C07281=1079.197,-43.335,442.916,173.632,20.227,153.492
C07282=1079.203,-43.085,442.903,173.633,20.229,153.493
C07283=1079.210,-42.836,442.891,173.635,20.230,153.493
C07284=1079.215,-42.586,442.879,173.636,20.232,153.493
C07285=1079.221,-42.337,442.866,173.637,20.234,153.493
C07286=1079.228,-42.087,442.854,173.639,20.236,153.493
C07287=1079.233,-41.837,442.842,173.640,20.238,153.493
C07288=1079.239,-41.588,442.830,173.642,20.240,153.493
C07289=1079.245,-41.338,442.817,173.644,20.242,153.493
C07290=1079.251,-41.088,442.805,173.645,20.244,153.494
C07291=1079.257,-40.839,442.793,173.646,20.246,153.494
C07292=1079.263,-40.589,442.780,173.648,20.248,153.494
C07293=1079.269,-40.340,442.769,173.649,20.250,153.494
C07294=1079.275,-40.090,442.756,173.650,20.252,153.494
C07295=1079.281,-39.840,442.743,173.652,20.253,153.494
C07296=1079.288,-39.590,442.731,173.653,20.255,153.494
C07297=1079.293,-39.341,442.719,173.655,20.258,153.494
C07298=1079.299,-39.091,442.707,173.657,20.260,153.495
C07299=1079.305,-38.842,442.694,173.658,20.262,153.495
C07300=1079.311,-38.592,442.682,173.659,20.263,153.495
C07301=1079.317,-38.342,442.670,173.661,20.265,153.495
C07302=1079.323,-38.093,442.657,173.662,20.267,153.495
C07303=1079.329,-37.843,442.645,173.663,20.269,153.495
C07304=1079.334,-37.593,442.632,173.665,20.272,153.495
C07305=1079.340,-37.343,442.620,173.667,20.274,153.496
C07306=1079.346,-37.094,442.608,173.668,20.276,153.496
C07307=1079.353,-36.845,442.595,173.669,20.278,153.496
C07308=1079.359,-36.595,442.582,173.671,20.279,153.496
C07309=1079.364,-36.345,442.570,173.672,20.281,153.496
C07310=1079.370,-36.096,442.558,173.673,20.283,153.496
C07311=1079.376,-35.846,442.545,173.674,20.285,153.496
C07312=1079.382,-35.596,442.533,173.677,20.288,153.497
C07313=1079.388,-35.347,442.520,173.678,20.290,153.497
C07314=1079.393,-35.097,442.507,173.679,20.292,153.497
C07315=1079.399,-34.848,442.495,173.680,20.294,153.497
C07316=1079.406,-34.599,442.483,173.682,20.296,153.497
C07317=1079.412,-34.349,442.470,173.683,20.298,153.497
C07318=1079.417,-34.099,442.457,173.685,20.300,153.497
C07319=1079.423,-33.849,442.445,173.687,20.302,153.498
C07320=1079.430,-33.575,442.431,173.688,20.304,153.498
C07321=1079.436,-33.302,442.417,173.689,20.306,153.498
C07322=1079.442,-33.028,442.404,173.691,20.309,153.498
C07323=1079.449,-32.754,442.390,173.692,20.311,153.498
C07324=1079.455,-32.504,442.376,173.694,20.313,153.499
C07325=1079.461,-32.254,442.364,173.695,20.315,153.499
C07326=1079.467,-32.004,442.351,173.697,20.317,153.499
C07327=1079.473,-31.755,442.339,173.699,20.318,153.499
C07328=1079.479,-31.505,442.325,173.700,20.320,153.499
C07329=1079.484,-31.256,442.313,173.701,20.322,153.499
C07330=1079.491,-31.007,442.301,173.703,20.324,153.499
C07331=1079.497,-30.757,442.288,173.704,20.326,153.500
C07332=1079.503,-30.507,442.275,173.705,20.328,153.500
C07333=1079.509,-30.258,442.263,173.707,20.331,153.500
C07334=1079.515,-30.008,442.250,173.709,20.333,153.500
C07335=1079.521,-29.758,442.237,173.710,20.335,153.500
C07336=1079.527,-29.509,442.225,173.711,20.337,153.500
C07337=1079.532,-29.259,442.212,173.712,20.339,153.500
C07338=1079.538,-29.010,442.199,173.714,20.341,153.501
C07339=1079.544,-28.760,442.187,173.716,20.343,153.501
C07340=1079.550,-28.510,442.174,173.717,20.345,153.501
C07341=1079.556,-28.261,442.161,173.719,20.347,153.501
C07342=1079.562,-28.011,442.148,173.720,20.349,153.501
C07343=1079.568,-27.761,442.136,173.721,20.351,153.501
C07344=1079.574,-27.512,442.122,173.722,20.353,153.501
C07345=1079.580,-27.262,442.110,173.725,20.355,153.502
C07346=1079.587,-27.013,442.097,173.726,20.357,153.502
C07347=1079.592,-26.763,442.084,173.727,20.359,153.502
C07348=1079.598,-26.513,442.071,173.728,20.361,153.502
C07349=1079.604,-26.264,442.058,173.730,20.363,153.502
C07350=1079.609,-26.014,442.045,173.731,20.365,153.502
C07351=1079.615,-25.765,442.032,173.733,20.368,153.503
C07352=1079.621,-25.515,442.020,173.734,20.370,153.503
C07353=1079.627,-25.266,442.006,173.736,20.372,153.503
C07354=1079.633,-25.016,441.994,173.737,20.374,153.503
C07355=1079.639,-24.766,441.981,173.738,20.376,153.503
C07356=1079.645,-24.517,441.967,173.739,20.378,153.504
C07357=1079.651,-24.267,441.955,173.742,20.381,153.504
C07358=1079.657,-24.017,441.941,173.743,20.383,153.504
C07359=1079.663,-23.768,441.929,173.744,20.385,153.504
C07360=1079.668,-23.518,441.915,173.745,20.387,153.504
C07361=1079.674,-23.268,441.903,173.747,20.389,153.504
C07362=1079.680,-23.020,441.890,173.748,20.391,153.504
C07363=1079.686,-22.770,441.877,173.750,20.393,153.505
C07364=1079.692,-22.520,441.864,173.751,20.395,153.505
C07365=1079.697,-22.270,441.851,173.753,20.397,153.505
C07366=1079.703,-22.021,441.837,173.754,20.399,153.505
C07367=1079.709,-21.771,441.825,173.755,20.401,153.505
C07368=1079.715,-21.522,441.812,173.757,20.403,153.505
C07369=1079.722,-21.273,441.798,173.759,20.405,153.506
C07370=1079.727,-21.022,441.785,173.760,20.407,153.506
C07371=1079.733,-20.773,441.772,173.761,20.409,153.506
C07372=1079.739,-20.523,441.759,173.763,20.411,153.506
C07373=1079.745,-20.274,441.746,173.764,20.413,153.506
C07374=1079.751,-20.024,441.732,173.766,20.416,153.507
C07375=1079.757,-19.774,441.720,173.767,20.418,153.507
C07376=1079.763,-19.525,441.706,173.768,20.420,153.507
C07377=1079.769,-19.275,441.694,173.770,20.422,153.507
C07378=1079.774,-19.026,441.680,173.771,20.424,153.507
C07379=1079.780,-18.776,441.667,173.772,20.426,153.507
C07380=1079.786,-18.527,441.654,173.774,20.429,153.507
C07381=1079.792,-18.277,441.641,173.776,20.431,153.508
C07382=1079.798,-18.028,441.627,173.777,20.433,153.508
C07383=1079.804,-17.778,441.614,173.778,20.435,153.508
C07384=1079.811,-17.503,441.600,173.780,20.437,153.508
C07385=1079.817,-17.228,441.585,173.782,20.440,153.508
C07386=1079.824,-16.953,441.570,173.783,20.442,153.509
C07387=1079.830,-16.679,441.557,173.785,20.444,153.509
C07388=1079.837,-16.429,441.543,173.786,20.446,153.509
C07389=1079.842,-16.180,441.529,173.788,20.448,153.509
C07390=1079.849,-15.930,441.516,173.789,20.450,153.509
C07391=1079.854,-15.680,441.503,173.791,20.453,153.509
C07392=1079.860,-15.431,441.489,173.792,20.455,153.510
C07393=1079.866,-15.182,441.476,173.793,20.457,153.510
C07394=1079.872,-14.932,441.463,173.795,20.459,153.510
C07395=1079.878,-14.682,441.450,173.796,20.461,153.510
C07396=1079.884,-14.433,441.436,173.797,20.463,153.510
C07397=1079.889,-14.183,441.423,173.799,20.465,153.510
C07398=1079.895,-13.934,441.409,173.800,20.468,153.511
C07399=1079.901,-13.684,441.396,173.802,20.470,153.511
C07400=1079.907,-13.435,441.383,173.803,20.472,153.511
C07401=1079.913,-13.185,441.370,173.804,20.474,153.511
C07402=1079.919,-12.936,441.356,173.806,20.476,153.511
C07403=1079.925,-12.686,441.342,173.808,20.478,153.512
C07404=1079.930,-12.436,441.329,173.809,20.481,153.512
C07405=1079.936,-12.187,441.316,173.810,20.483,153.512
C07406=1079.942,-11.937,441.302,173.811,20.485,153.512
C07407=1079.948,-11.687,441.289,173.814,20.487,153.512
C07408=1079.954,-11.438,441.275,173.815,20.489,153.512
C07409=1079.960,-11.189,441.261,173.816,20.491,153.513
C07410=1079.965,-10.938,441.248,173.817,20.494,153.513
C07411=1079.972,-10.689,441.235,173.819,20.496,153.513
C07412=1079.977,-10.440,441.221,173.821,20.498,153.513
C07413=1079.983,-10.190,441.208,173.822,20.500,153.513
C07414=1079.989,-9.941,441.194,173.823,20.502,153.514
C07415=1079.995,-9.691,441.181,173.825,20.504,153.514
C07416=1080.001,-9.441,441.166,173.826,20.507,153.514
C07417=1080.007,-9.192,441.153,173.828,20.509,153.514
C07418=1080.013,-8.942,441.139,173.829,20.511,153.514
C07419=1080.019,-8.693,441.126,173.830,20.513,153.515
C07420=1080.024,-8.443,441.113,173.832,20.515,153.515
C07421=1080.030,-8.193,441.099,173.833,20.517,153.515
C07422=1080.036,-7.944,441.086,173.835,20.520,153.515
C07423=1080.042,-7.694,441.072,173.836,20.522,153.515
C07424=1080.048,-7.445,441.058,173.837,20.524,153.515
C07425=1080.053,-7.195,441.044,173.839,20.526,153.516
C07426=1080.060,-6.946,441.031,173.840,20.528,153.516
C07427=1080.065,-6.696,441.017,173.842,20.530,153.516
C07428=1080.071,-6.447,441.004,173.843,20.533,153.516
C07429=1080.077,-6.197,440.990,173.845,20.535,153.516
C07430=1080.084,-5.947,440.976,173.846,20.537,153.517
C07431=1080.089,-5.698,440.963,173.848,20.539,153.517
C07432=1080.095,-5.448,440.949,173.849,20.541,153.517
C07433=1080.101,-5.199,440.936,173.850,20.544,153.517
C07434=1080.107,-4.949,440.921,173.852,20.546,153.517
C07435=1080.113,-4.699,440.908,173.853,20.548,153.517
C07436=1080.119,-4.450,440.894,173.855,20.550,153.518
C07437=1080.125,-4.201,440.880,173.856,20.552,153.518
C07438=1080.131,-3.952,440.866,173.858,20.554,153.518
C07439=1080.137,-3.701,440.852,173.859,20.557,153.518
C07440=1080.143,-3.452,440.839,173.860,20.559,153.518
C07441=1080.148,-3.202,440.825,173.862,20.561,153.519
C07442=1080.154,-2.953,440.811,173.864,20.563,153.519
C07443=1080.160,-2.704,440.798,173.865,20.566,153.519
C07444=1080.166,-2.453,440.784,173.866,20.568,153.519
C07445=1080.172,-2.204,440.770,173.868,20.570,153.519
C07446=1080.177,-1.954,440.756,173.869,20.572,153.519
C07447=1080.183,-1.705,440.741,173.871,20.575,153.520
C07448=1080.190,-1.429,440.727,173.872,20.577,153.520
C07449=1080.196,-1.153,440.711,173.874,20.580,153.520
C07450=1080.202,-0.875,440.695,173.875,20.582,153.520
C07451=1080.209,-0.600,440.680,173.877,20.585,153.521
C07452=1080.215,-0.350,440.666,173.878,20.587,153.521
C07453=1080.220,-0.100,440.652,173.880,20.589,153.521
C07454=1080.226,0.148,440.638,173.881,20.591,153.521
C07455=1080.232,0.399,440.624,173.883,20.593,153.521
C07456=1080.237,0.648,440.610,173.884,20.595,153.522
C07457=1080.244,0.898,440.597,173.885,20.598,153.522
C07458=1080.249,1.147,440.583,173.887,20.600,153.522
C07459=1080.255,1.396,440.568,173.889,20.602,153.522
C07460=1080.261,1.646,440.554,173.890,20.604,153.522
C07461=1080.266,1.896,440.540,173.891,20.607,153.523
C07462=1080.272,2.146,440.526,173.892,20.609,153.523
C07463=1080.278,2.395,440.512,173.894,20.611,153.523
C07464=1080.284,2.644,440.498,173.896,20.614,153.523
C07465=1080.290,2.894,440.484,173.897,20.616,153.523
C07466=1080.296,3.143,440.469,173.898,20.618,153.524
C07467=1080.301,3.393,440.456,173.900,20.620,153.524
C07468=1080.307,3.643,440.441,173.901,20.623,153.524
C07469=1080.313,3.892,440.428,173.903,20.625,153.524
C07470=1080.319,4.141,440.413,173.904,20.627,153.524
C07471=1080.324,4.391,440.399,173.905,20.629,153.525
C07472=1080.331,4.641,440.385,173.907,20.632,153.525
C07473=1080.337,4.890,440.371,173.909,20.634,153.525
C07474=1080.342,5.139,440.357,173.910,20.636,153.525
C07475=1080.348,5.390,440.343,173.911,20.638,153.525
C07476=1080.354,5.639,440.328,173.913,20.641,153.526
C07477=1080.359,5.888,440.314,173.914,20.643,153.526
C07478=1080.366,6.138,440.299,173.916,20.644,153.526
C07479=1080.371,6.388,440.286,173.917,20.647,153.526
C07480=1080.377,6.637,440.272,173.918,20.649,153.526
C07481=1080.383,6.887,440.257,173.920,20.651,153.527
C07482=1080.389,7.136,440.243,173.921,20.654,153.527
C07483=1080.395,7.385,440.229,173.923,20.656,153.527
C07484=1080.401,7.635,440.215,173.924,20.658,153.527
C07485=1080.407,7.885,440.201,173.926,20.660,153.527
C07486=1080.413,8.134,440.186,173.927,20.663,153.528
C07487=1080.419,8.384,440.172,173.929,20.665,153.528
C07488=1080.424,8.633,440.157,173.930,20.667,153.528
C07489=1080.430,8.883,440.144,173.932,20.669,153.528
C07490=1080.436,9.132,440.129,173.933,20.672,153.528
C07491=1080.442,9.382,440.115,173.934,20.674,153.529
C07492=1080.447,9.631,440.100,173.936,20.676,153.529
C07493=1080.454,9.881,440.086,173.938,20.678,153.529
C07494=1080.459,10.130,440.071,173.939,20.681,153.529
C07495=1080.465,10.380,440.057,173.940,20.683,153.529
C07496=1080.471,10.629,440.042,173.942,20.685,153.530
C07497=1080.477,10.879,440.029,173.944,20.687,153.530
C07498=1080.483,11.128,440.014,173.945,20.690,153.530
C07499=1080.489,11.378,440.000,173.946,20.691,153.530
C07500=1080.496,11.627,439.985,173.947,20.693,153.530
C07501=1080.501,11.877,439.972,173.949,20.695,153.530
C07502=1080.508,12.127,439.957,173.951,20.698,153.531
C07503=1080.513,12.376,439.943,173.952,20.700,153.531
C07504=1080.519,12.625,439.928,173.953,20.702,153.531
C07505=1080.525,12.875,439.913,173.955,20.704,153.531
C07506=1080.531,13.124,439.899,173.957,20.707,153.532
C07507=1080.537,13.374,439.884,173.958,20.709,153.532
C07508=1080.542,13.624,439.871,173.959,20.711,153.532
C07509=1080.549,13.873,439.856,173.960,20.713,153.532
C07510=1080.555,14.122,439.841,173.962,20.716,153.532
C07511=1080.561,14.372,439.827,173.964,20.718,153.532
C07512=1080.566,14.650,439.811,173.965,20.720,153.533
C07513=1080.573,14.929,439.794,173.967,20.723,153.533
C07514=1080.579,15.207,439.778,173.969,20.726,153.533
C07515=1080.586,15.485,439.762,173.970,20.728,153.533
C07516=1080.592,15.735,439.747,173.971,20.731,153.534
C07517=1080.598,15.984,439.732,173.974,20.733,153.534
C07518=1080.604,16.234,439.718,173.975,20.735,153.534
C07519=1080.610,16.483,439.703,173.976,20.737,153.534
C07520=1080.615,16.732,439.689,173.977,20.739,153.534
C07521=1080.621,16.983,439.674,173.979,20.742,153.535
C07522=1080.626,17.232,439.659,173.980,20.744,153.535
C07523=1080.633,17.482,439.644,173.982,20.746,153.535
C07524=1080.639,17.730,439.630,173.983,20.748,153.535
C07525=1080.645,17.981,439.615,173.985,20.751,153.535
C07526=1080.650,18.230,439.600,173.986,20.753,153.536
C07527=1080.656,18.480,439.585,173.988,20.755,153.536
C07528=1080.662,18.729,439.571,173.989,20.757,153.536
C07529=1080.668,18.979,439.556,173.991,20.760,153.536
C07530=1080.674,19.228,439.542,173.992,20.762,153.536
C07531=1080.679,19.478,439.526,173.994,20.764,153.537
C07532=1080.685,19.727,439.512,173.995,20.767,153.537
C07533=1080.692,19.976,439.497,173.997,20.769,153.537
C07534=1080.697,20.226,439.483,173.998,20.771,153.537
C07535=1080.703,20.476,439.467,173.999,20.773,153.537
C07536=1080.708,20.725,439.453,174.001,20.776,153.538
C07537=1080.714,20.974,439.438,174.003,20.778,153.538
C07538=1080.720,21.224,439.423,174.004,20.780,153.538
C07539=1080.725,21.473,439.409,174.005,20.782,153.538
C07540=1080.732,21.723,439.394,174.007,20.785,153.538
C07541=1080.737,21.972,439.379,174.008,20.787,153.539
C07542=1080.743,22.222,439.364,174.010,20.789,153.539
C07543=1080.749,22.471,439.349,174.011,20.791,153.539
C07544=1080.755,22.721,439.334,174.013,20.794,153.539
C07545=1080.760,22.970,439.319,174.014,20.796,153.539
C07546=1080.767,23.220,439.304,174.016,20.798,153.540
C07547=1080.772,23.470,439.289,174.017,20.801,153.540
C07548=1080.778,23.719,439.275,174.019,20.803,153.540
C07549=1080.784,23.969,439.260,174.020,20.805,153.540
C07550=1080.789,24.218,439.245,174.021,20.808,153.541
C07551=1080.796,24.468,439.230,174.023,20.810,153.541
C07552=1080.801,24.717,439.215,174.025,20.812,153.541
C07553=1080.807,24.967,439.200,174.026,20.814,153.541
C07554=1080.813,25.216,439.185,174.027,20.816,153.541
C07555=1080.819,25.466,439.169,174.029,20.819,153.541
C07556=1080.824,25.714,439.155,174.031,20.821,153.542
C07557=1080.831,25.964,439.140,174.032,20.823,153.542
C07558=1080.836,26.214,439.124,174.034,20.826,153.542
C07559=1080.842,26.463,439.110,174.035,20.828,153.542
C07560=1080.849,26.713,439.095,174.036,20.830,153.543
C07561=1080.854,26.962,439.080,174.038,20.832,153.543
C07562=1080.860,27.212,439.065,174.040,20.835,153.543
C07563=1080.866,27.462,439.049,174.041,20.837,153.543
C07564=1080.871,27.711,439.035,174.042,20.839,153.543
C07565=1080.877,27.961,439.019,174.043,20.841,153.544
C07566=1080.883,28.209,439.004,174.045,20.844,153.544
C07567=1080.889,28.459,438.990,174.047,20.846,153.544
C07568=1080.895,28.708,438.974,174.048,20.848,153.544
C07569=1080.901,28.957,438.959,174.050,20.850,153.544
C07570=1080.907,29.207,438.943,174.051,20.853,153.545
C07571=1080.912,29.457,438.928,174.053,20.855,153.545
C07572=1080.918,29.706,438.913,174.054,20.857,153.545
C07573=1080.923,29.956,438.898,174.056,20.860,153.545
C07574=1080.929,30.205,438.883,174.057,20.862,153.545
C07575=1080.935,30.455,438.867,174.058,20.864,153.546
C07576=1080.941,30.735,438.850,174.061,20.867,153.546
C07577=1080.948,31.014,438.833,174.063,20.870,153.546
C07578=1080.954,31.294,438.816,174.064,20.872,153.546
C07579=1080.961,31.574,438.799,174.066,20.874,153.546
C07580=1080.967,31.823,438.784,174.067,20.876,153.547
C07581=1080.972,32.073,438.769,174.068,20.879,153.547
C07582=1080.978,32.321,438.753,174.070,20.881,153.547
C07583=1080.984,32.571,438.738,174.072,20.883,153.547
C07584=1080.990,32.821,438.722,174.073,20.886,153.548
C07585=1080.995,33.070,438.708,174.074,20.888,153.548
C07586=1081.001,33.320,438.692,174.076,20.890,153.548
C07587=1081.008,33.569,438.676,174.077,20.893,153.548
C07588=1081.013,33.818,438.661,174.079,20.895,153.548
C07589=1081.019,34.068,438.646,174.081,20.897,153.548
C07590=1081.025,34.318,438.631,174.082,20.900,153.549
C07591=1081.030,34.567,438.615,174.083,20.902,153.549
C07592=1081.037,34.816,438.600,174.085,20.904,153.549
C07593=1081.042,35.066,438.584,174.087,20.906,153.549
C07594=1081.048,35.315,438.568,174.088,20.908,153.550
C07595=1081.054,35.565,438.554,174.089,20.910,153.550
C07596=1081.060,35.815,438.538,174.091,20.913,153.550
C07597=1081.065,36.064,438.523,174.093,20.915,153.550
C07598=1081.071,36.313,438.507,174.094,20.917,153.550
C07599=1081.077,36.563,438.492,174.096,20.920,153.550
C07600=1081.083,36.813,438.476,174.097,20.922,153.551
C07601=1081.089,37.061,438.461,174.098,20.924,153.551
C07602=1081.094,37.311,438.445,174.101,20.927,153.551
C07603=1081.100,37.561,438.430,174.102,20.929,153.551
C07604=1081.106,37.810,438.414,174.103,20.931,153.552
C07605=1081.112,38.059,438.399,174.104,20.933,153.552
C07606=1081.118,38.309,438.383,174.106,20.936,153.552
C07607=1081.123,38.559,438.367,174.108,20.938,153.552
C07608=1081.129,38.808,438.352,174.109,20.940,153.552
C07609=1081.135,39.057,438.336,174.111,20.943,153.553
C07610=1081.141,39.307,438.321,174.112,20.945,153.553
C07611=1081.146,39.556,438.305,174.114,20.947,153.553
C07612=1081.152,39.806,438.289,174.116,20.950,153.553
C07613=1081.158,40.055,438.274,174.117,20.952,153.553
C07614=1081.163,40.304,438.258,174.118,20.954,153.554
C07615=1081.169,40.554,438.243,174.120,20.957,153.554
C07616=1081.175,40.803,438.227,174.121,20.959,153.554
C07617=1081.181,41.053,438.211,174.123,20.960,153.554
C07618=1081.186,41.302,438.195,174.125,20.963,153.554
C07619=1081.192,41.552,438.180,174.126,20.965,153.555
C07620=1081.198,41.801,438.164,174.127,20.967,153.555
C07621=1081.204,42.051,438.148,174.129,20.970,153.555
C07622=1081.209,42.300,438.133,174.131,20.972,153.555
C07623=1081.215,42.550,438.117,174.132,20.974,153.555
C07624=1081.221,42.799,438.101,174.134,20.977,153.556
C07625=1081.227,43.049,438.086,174.135,20.979,153.556
C07626=1081.233,43.298,438.070,174.137,20.981,153.556
C07627=1081.238,43.547,438.054,174.138,20.983,153.556
C07628=1081.244,43.796,438.038,174.140,20.986,153.556
C07629=1081.250,44.046,438.023,174.141,20.988,153.557
C07630=1081.256,44.296,438.006,174.143,20.990,153.557
C07631=1081.261,44.544,437.990,174.145,20.993,153.557
C07632=1081.267,44.794,437.975,174.146,20.995,153.557
C07633=1081.273,45.044,437.959,174.147,20.997,153.558
C07634=1081.278,45.293,437.943,174.149,21.000,153.558
C07635=1081.284,45.542,437.927,174.150,21.002,153.558
C07636=1081.290,45.792,437.911,174.152,21.004,153.558
C07637=1081.295,46.042,437.895,174.154,21.007,153.558
C07638=1081.301,46.291,437.879,174.155,21.009,153.558
C07639=1081.306,46.540,437.864,174.156,21.011,153.559
C07640=1081.313,46.820,437.845,174.158,21.013,153.559
C07641=1081.319,47.100,437.828,174.160,21.016,153.559
C07642=1081.326,47.380,437.810,174.161,21.019,153.559
C07643=1081.331,47.660,437.792,174.164,21.021,153.560
C07644=1081.337,47.909,437.776,174.165,21.024,153.560
C07645=1081.343,48.158,437.759,174.167,21.026,153.560
C07646=1081.349,48.408,437.744,174.168,21.028,153.560
C07647=1081.354,48.657,437.728,174.169,21.031,153.561
C07648=1081.360,48.906,437.712,174.172,21.033,153.561
C07649=1081.366,49.156,437.695,174.173,21.035,153.561
C07650=1081.372,49.406,437.680,174.174,21.037,153.561
C07651=1081.378,49.655,437.664,174.176,21.040,153.561
C07652=1081.384,49.904,437.647,174.178,21.042,153.561
C07653=1081.389,50.153,437.631,174.179,21.044,153.562
C07654=1081.394,50.403,437.615,174.181,21.047,153.562
C07655=1081.400,50.653,437.599,174.182,21.049,153.562
C07656=1081.406,50.902,437.583,174.183,21.051,153.562
C07657=1081.412,51.151,437.566,174.185,21.054,153.562
C07658=1081.418,51.401,437.550,174.187,21.056,153.563
C07659=1081.423,51.651,437.535,174.188,21.057,153.563
C07660=1081.429,51.899,437.519,174.190,21.060,153.563
C07661=1081.435,52.149,437.503,174.191,21.062,153.563
C07662=1081.441,52.398,437.486,174.193,21.064,153.563
C07663=1081.446,52.648,437.469,174.195,21.067,153.564
C07664=1081.451,52.898,437.454,174.196,21.069,153.564
C07665=1081.457,53.147,437.438,174.198,21.072,153.564
C07666=1081.463,53.396,437.421,174.200,21.074,153.564
C07667=1081.469,53.646,437.405,174.201,21.076,153.565
C07668=1081.475,53.895,437.389,174.203,21.078,153.565
C07669=1081.481,54.144,437.373,174.204,21.080,153.565
C07670=1081.486,54.393,437.356,174.205,21.083,153.565
C07671=1081.492,54.643,437.340,174.208,21.085,153.565
C07672=1081.498,54.892,437.324,174.209,21.087,153.565
C07673=1081.503,55.142,437.308,174.210,21.089,153.566
C07674=1081.509,55.391,437.292,174.212,21.092,153.566
C07675=1081.515,55.641,437.276,174.213,21.094,153.566
C07676=1081.520,55.890,437.259,174.215,21.096,153.566
C07677=1081.526,56.140,437.242,174.217,21.098,153.566
C07678=1081.532,56.389,437.226,174.218,21.100,153.567
C07679=1081.538,56.638,437.210,174.220,21.103,153.567
C07680=1081.544,56.888,437.194,174.222,21.105,153.567
C07681=1081.550,57.137,437.177,174.223,21.107,153.567
C07682=1081.555,57.387,437.161,174.225,21.110,153.567
C07683=1081.561,57.636,437.144,174.226,21.112,153.568
C07684=1081.567,57.885,437.128,174.228,21.114,153.568
C07685=1081.573,58.135,437.112,174.230,21.117,153.568
C07686=1081.579,58.384,437.095,174.231,21.118,153.568
C07687=1081.584,58.634,437.079,174.232,21.120,153.568
C07688=1081.590,58.883,437.062,174.235,21.123,153.568
C07689=1081.596,59.132,437.046,174.236,21.125,153.569
C07690=1081.602,59.382,437.030,174.238,21.128,153.569
C07691=1081.608,59.631,437.013,174.239,21.130,153.569
C07692=1081.614,59.880,436.996,174.241,21.132,153.569
C07693=1081.620,60.129,436.980,174.243,21.134,153.569
C07694=1081.626,60.379,436.964,174.244,21.137,153.570
C07695=1081.631,60.628,436.947,174.245,21.138,153.570
C07696=1081.637,60.878,436.930,174.247,21.141,153.570
C07697=1081.643,61.127,436.914,174.249,21.143,153.570
C07698=1081.649,61.377,436.898,174.250,21.145,153.570
C07699=1081.654,61.626,436.881,174.252,21.147,153.570
C07700=1081.660,61.876,436.865,174.254,21.149,153.571
C07701=1081.666,62.124,436.848,174.256,21.152,153.571
C07702=1081.672,62.374,436.832,174.257,21.154,153.571
C07703=1081.677,62.623,436.815,174.258,21.156,153.571
C07704=1081.684,62.903,436.796,174.261,21.158,153.571
C07705=1081.692,63.182,436.778,174.262,21.161,153.572
C07706=1081.698,63.462,436.759,174.264,21.163,153.572
C07707=1081.704,63.741,436.741,174.266,21.166,153.572
C07708=1081.710,63.991,436.724,174.267,21.168,153.572
C07709=1081.716,64.240,436.708,174.269,21.171,153.572
C07710=1081.722,64.490,436.691,174.271,21.172,153.572
C07711=1081.728,64.739,436.673,174.273,21.175,153.573
C07712=1081.734,64.988,436.657,174.274,21.177,153.573
C07713=1081.739,65.238,436.640,174.276,21.179,153.573
C07714=1081.745,65.487,436.624,174.278,21.182,153.573
C07715=1081.750,65.737,436.606,174.279,21.184,153.573
C07716=1081.756,65.986,436.590,174.280,21.186,153.574
C07717=1081.762,66.235,436.574,174.282,21.188,153.574
C07718=1081.767,66.485,436.557,174.284,21.190,153.574
C07719=1081.774,66.734,436.540,174.286,21.192,153.574
C07720=1081.779,66.983,436.523,174.287,21.195,153.574
C07721=1081.785,67.233,436.507,174.288,21.197,153.575
C07722=1081.790,67.482,436.489,174.291,21.199,153.575
C07723=1081.797,67.732,436.473,174.292,21.201,153.575
C07724=1081.802,67.981,436.456,174.294,21.204,153.575
C07725=1081.808,68.230,436.439,174.295,21.206,153.575
C07726=1081.814,68.480,436.422,174.297,21.208,153.575
C07727=1081.819,68.729,436.405,174.299,21.210,153.576
C07728=1081.825,68.978,436.388,174.300,21.212,153.576
C07729=1081.830,69.228,436.371,174.302,21.215,153.576
C07730=1081.837,69.477,436.354,174.304,21.217,153.576
C07731=1081.842,69.726,436.338,174.305,21.219,153.576
C07732=1081.848,69.976,436.321,174.307,21.222,153.577
C07733=1081.854,70.225,436.303,174.308,21.223,153.577
C07734=1081.860,70.475,436.287,174.311,21.226,153.577
C07735=1081.865,70.724,436.270,174.312,21.228,153.577
C07736=1081.871,70.973,436.253,174.313,21.230,153.577
C07737=1081.877,71.222,436.236,174.315,21.232,153.577
C07738=1081.882,71.472,436.219,174.317,21.235,153.578
C07739=1081.887,71.721,436.201,174.319,21.237,153.578
C07740=1081.894,71.971,436.185,174.320,21.239,153.578
C07741=1081.900,72.220,436.167,174.321,21.241,153.578
C07742=1081.905,72.470,436.150,174.324,21.243,153.578
C07743=1081.911,72.718,436.133,174.325,21.245,153.578
C07744=1081.916,72.968,436.116,174.327,21.248,153.579
C07745=1081.922,73.217,436.099,174.328,21.250,153.579
C07746=1081.928,73.466,436.083,174.330,21.252,153.579
C07747=1081.934,73.716,436.065,174.332,21.255,153.579
C07748=1081.939,73.966,436.048,174.333,21.256,153.579
C07749=1081.945,74.214,436.031,174.335,21.259,153.579
C07750=1081.951,74.464,436.014,174.337,21.261,153.580
C07751=1081.956,74.713,435.996,174.339,21.263,153.580
C07752=1081.962,74.963,435.979,174.340,21.266,153.580
C07753=1081.968,75.212,435.962,174.341,21.268,153.580
C07754=1081.974,75.461,435.945,174.344,21.270,153.580
C07755=1081.979,75.711,435.928,174.345,21.272,153.581
C07756=1081.985,75.960,435.911,174.347,21.274,153.581
C07757=1081.991,76.210,435.894,174.348,21.276,153.581
C07758=1081.996,76.459,435.876,174.350,21.278,153.581
C07759=1082.002,76.708,435.859,174.352,21.281,153.581
C07760=1082.008,76.957,435.842,174.353,21.283,153.581
C07761=1082.013,77.206,435.825,174.356,21.285,153.581
C07762=1082.020,77.456,435.807,174.357,21.287,153.582
C07763=1082.025,77.706,435.790,174.359,21.290,153.582
C07764=1082.031,77.955,435.773,174.360,21.292,153.582
C07765=1082.037,78.204,435.755,174.362,21.294,153.582
C07766=1082.042,78.454,435.738,174.364,21.296,153.582
C07767=1082.048,78.703,435.721,174.365,21.298,153.583
C07768=1082.055,78.982,435.701,174.367,21.300,153.583
C07769=1082.061,79.262,435.682,174.369,21.303,153.583
C07770=1082.067,79.541,435.662,174.371,21.305,153.583
C07771=1082.073,79.821,435.643,174.373,21.308,153.583
C07772=1082.079,80.070,435.626,174.375,21.311,153.584
C07773=1082.085,80.319,435.608,174.376,21.313,153.584
C07774=1082.091,80.568,435.590,174.378,21.315,153.584
C07775=1082.096,80.818,435.573,174.380,21.317,153.584
C07776=1082.101,81.067,435.556,174.381,21.319,153.584
C07777=1082.107,81.317,435.538,174.383,21.321,153.584
C07778=1082.113,81.566,435.520,174.385,21.323,153.585
C07779=1082.118,81.815,435.503,174.387,21.326,153.585
C07780=1082.124,82.065,435.486,174.388,21.328,153.585
C07781=1082.130,82.314,435.468,174.390,21.330,153.585
C07782=1082.135,82.563,435.450,174.392,21.332,153.585
C07783=1082.141,82.812,435.433,174.393,21.334,153.585
C07784=1082.147,83.062,435.415,174.395,21.337,153.586
C07785=1082.152,83.311,435.397,174.396,21.339,153.586
C07786=1082.158,83.561,435.380,174.399,21.341,153.586
C07787=1082.163,83.810,435.363,174.400,21.343,153.586
C07788=1082.169,84.060,435.345,174.402,21.345,153.586
C07789=1082.176,84.308,435.328,174.403,21.347,153.586
C07790=1082.181,84.557,435.310,174.406,21.350,153.587
C07791=1082.187,84.807,435.292,174.407,21.352,153.587
C07792=1082.193,85.056,435.275,174.408,21.354,153.587
C07793=1082.198,85.305,435.257,174.411,21.356,153.587
C07794=1082.204,85.555,435.239,174.412,21.358,153.587
C07795=1082.210,85.804,435.222,174.414,21.360,153.587
C07796=1082.215,86.053,435.204,174.415,21.362,153.588
C07797=1082.221,86.303,435.186,174.418,21.365,153.588
C07798=1082.227,86.552,435.169,174.419,21.367,153.588
C07799=1082.233,86.801,435.151,174.421,21.369,153.588
C07800=1082.238,87.051,435.133,174.423,21.371,153.588
C07801=1082.243,87.300,435.115,174.425,21.373,153.588
C07802=1082.249,87.549,435.098,174.426,21.375,153.588
C07803=1082.255,87.799,435.080,174.428,21.378,153.589
C07804=1082.261,88.048,435.062,174.430,21.380,153.589
C07805=1082.267,88.297,435.044,174.431,21.382,153.589
C07806=1082.272,88.546,435.027,174.433,21.384,153.589
C07807=1082.278,88.796,435.009,174.435,21.386,153.589
C07808=1082.284,89.045,434.991,174.437,21.388,153.589
C07809=1082.289,89.294,434.973,174.438,21.390,153.590
C07810=1082.295,89.544,434.956,174.440,21.393,153.590
C07811=1082.301,89.793,434.938,174.442,21.395,153.590
C07812=1082.307,90.042,434.920,174.444,21.397,153.590
C07813=1082.313,90.292,434.902,174.445,21.399,153.590
C07814=1082.318,90.541,434.885,174.448,21.401,153.590
C07815=1082.324,90.791,434.867,174.449,21.403,153.590
C07816=1082.330,91.039,434.849,174.451,21.405,153.590
C07817=1082.335,91.289,434.830,174.453,21.407,153.591
C07818=1082.341,91.538,434.813,174.455,21.409,153.591
C07819=1082.347,91.787,434.795,174.456,21.411,153.591
C07820=1082.353,92.037,434.777,174.457,21.413,153.591
C07821=1082.357,92.286,434.759,174.460,21.416,153.591
C07822=1082.364,92.536,434.741,174.461,21.418,153.591
C07823=1082.369,92.784,434.723,174.463,21.420,153.592
C07824=1082.375,93.033,434.705,174.465,21.422,153.592
C07825=1082.380,93.284,434.687,174.467,21.424,153.592
C07826=1082.386,93.533,434.669,174.468,21.426,153.592
C07827=1082.392,93.782,434.651,174.470,21.429,153.592
C07828=1082.398,94.031,434.633,174.472,21.431,153.592
C07829=1082.403,94.280,434.615,174.474,21.433,153.593
C07830=1082.409,94.530,434.597,174.475,21.435,153.593
C07831=1082.414,94.779,434.579,174.478,21.437,153.593
C07832=1082.421,95.059,434.558,174.480,21.440,153.593
C07833=1082.428,95.338,434.538,174.481,21.442,153.593
C07834=1082.434,95.617,434.518,174.483,21.444,153.593
C07835=1082.440,95.897,434.497,174.485,21.447,153.594
C07836=1082.445,96.146,434.480,174.487,21.449,153.594
C07837=1082.452,96.395,434.461,174.489,21.451,153.594
C07838=1082.456,96.644,434.443,174.490,21.453,153.594
C07839=1082.462,96.894,434.425,174.493,21.455,153.594
C07840=1082.468,97.142,434.407,174.494,21.457,153.594
C07841=1082.474,97.393,434.388,174.496,21.459,153.594
C07842=1082.479,97.642,434.370,174.498,21.461,153.595
C07843=1082.486,97.891,434.352,174.500,21.464,153.595
C07844=1082.490,98.140,434.334,174.501,21.466,153.595
C07845=1082.496,98.390,434.316,174.503,21.468,153.595
C07846=1082.503,98.639,434.297,174.505,21.470,153.595
C07847=1082.508,98.888,434.279,174.507,21.472,153.595
C07848=1082.514,99.137,434.260,174.508,21.474,153.595
C07849=1082.520,99.386,434.243,174.511,21.476,153.596
C07850=1082.525,99.637,434.224,174.512,21.478,153.596
C07851=1082.531,99.885,434.206,174.514,21.480,153.596
C07852=1082.537,100.135,434.188,174.516,21.482,153.596
C07853=1082.542,100.383,434.169,174.518,21.485,153.596
C07854=1082.548,100.633,434.151,174.519,21.486,153.596
C07855=1082.554,100.882,434.133,174.522,21.488,153.596
C07856=1082.559,101.132,434.114,174.523,21.490,153.596
C07857=1082.566,101.381,434.096,174.525,21.493,153.597
C07858=1082.571,101.630,434.078,174.526,21.495,153.597
C07859=1082.577,101.879,434.059,174.529,21.497,153.597
C07860=1082.582,102.129,434.041,174.531,21.499,153.597
C07861=1082.588,102.378,434.022,174.532,21.501,153.597
C07862=1082.593,102.627,434.004,174.535,21.503,153.597
C07863=1082.599,102.876,433.985,174.536,21.505,153.597
C07864=1082.604,103.125,433.967,174.538,21.508,153.598
C07865=1082.610,103.375,433.948,174.540,21.509,153.598
C07866=1082.615,103.624,433.930,174.542,21.512,153.598
C07867=1082.621,103.873,433.911,174.543,21.514,153.598
C07868=1082.627,104.123,433.892,174.545,21.516,153.598
C07869=1082.632,104.372,433.874,174.547,21.518,153.598
C07870=1082.639,104.621,433.856,174.549,21.520,153.598
C07871=1082.643,104.870,433.837,174.551,21.522,153.599
C07872=1082.649,105.120,433.818,174.553,21.524,153.599
C07873=1082.655,105.368,433.800,174.554,21.526,153.599
C07874=1082.660,105.618,433.781,174.556,21.529,153.599
C07875=1082.667,105.867,433.763,174.558,21.531,153.599
C07876=1082.672,106.116,433.744,174.560,21.532,153.599
C07877=1082.677,106.366,433.725,174.561,21.534,153.599
C07878=1082.683,106.615,433.707,174.564,21.537,153.600
C07879=1082.689,106.864,433.688,174.566,21.539,153.600
C07880=1082.695,107.114,433.670,174.567,21.541,153.600
C07881=1082.700,107.362,433.651,174.570,21.543,153.600
C07882=1082.706,107.612,433.632,174.571,21.545,153.600
C07883=1082.712,107.861,433.613,174.573,21.547,153.600
C07884=1082.717,108.110,433.595,174.575,21.549,153.600
C07885=1082.723,108.360,433.576,174.577,21.551,153.600
C07886=1082.729,108.609,433.557,174.578,21.553,153.601
C07887=1082.734,108.858,433.538,174.581,21.555,153.601
C07888=1082.740,109.107,433.520,174.582,21.557,153.601
C07889=1082.746,109.357,433.501,174.584,21.560,153.601
C07890=1082.751,109.606,433.482,174.586,21.561,153.601
C07891=1082.757,109.855,433.463,174.588,21.563,153.601
C07892=1082.763,110.105,433.445,174.590,21.566,153.601
C07893=1082.768,110.353,433.426,174.592,21.567,153.601
C07894=1082.774,110.603,433.407,174.594,21.570,153.601
C07895=1082.780,110.852,433.388,174.595,21.571,153.602
C07896=1082.786,111.131,433.367,174.598,21.574,153.602
C07897=1082.793,111.411,433.346,174.600,21.576,153.602
C07898=1082.799,111.690,433.325,174.602,21.579,153.602
C07899=1082.806,111.970,433.304,174.604,21.581,153.602
C07900=1082.812,112.219,433.284,174.606,21.582,153.602
C07901=1082.816,112.469,433.266,174.608,21.585,153.602
C07902=1082.822,112.718,433.247,174.609,21.587,153.603
C07903=1082.828,112.967,433.228,174.612,21.589,153.603
C07904=1082.834,113.216,433.210,174.613,21.590,153.603
C07905=1082.839,113.465,433.190,174.615,21.593,153.603
C07906=1082.845,113.715,433.171,174.618,21.595,153.603
C07907=1082.851,113.964,433.152,174.619,21.597,153.603
C07908=1082.856,114.213,433.134,174.621,21.599,153.603
C07909=1082.862,114.462,433.114,174.623,21.601,153.603
C07910=1082.868,114.711,433.095,174.625,21.603,153.603
C07911=1082.873,114.960,433.076,174.627,21.605,153.604
C07912=1082.879,115.210,433.057,174.629,21.607,153.604
C07913=1082.884,115.459,433.038,174.631,21.609,153.604
C07914=1082.889,115.708,433.019,174.632,21.611,153.604
C07915=1082.895,115.957,433.000,174.635,21.614,153.604
C07916=1082.901,116.207,432.980,174.636,21.615,153.604
C07917=1082.906,116.456,432.961,174.638,21.618,153.604
C07918=1082.911,116.705,432.942,174.641,21.620,153.604
C07919=1082.917,116.954,432.923,174.642,21.622,153.605
C07920=1082.923,117.204,432.904,174.644,21.624,153.605
C07921=1082.929,117.453,432.884,174.646,21.626,153.605
C07922=1082.934,117.702,432.866,174.648,21.628,153.605
C07923=1082.939,117.951,432.846,174.649,21.630,153.605
C07924=1082.945,118.201,432.827,174.652,21.632,153.605
C07925=1082.950,118.449,432.808,174.654,21.634,153.605
C07926=1082.956,118.698,432.788,174.655,21.636,153.605
C07927=1082.962,118.948,432.769,174.658,21.638,153.606
C07928=1082.967,119.197,432.750,174.659,21.640,153.606
C07929=1082.973,119.447,432.731,174.661,21.642,153.606
C07930=1082.978,119.695,432.712,174.664,21.645,153.606
C07931=1082.984,119.945,432.692,174.665,21.646,153.606
C07932=1082.990,120.194,432.673,174.667,21.648,153.606
C07933=1082.996,120.443,432.653,174.669,21.650,153.606
C07934=1083.001,120.692,432.634,174.671,21.652,153.606
C07935=1083.006,120.941,432.615,174.673,21.654,153.606
C07936=1083.012,121.191,432.596,174.675,21.656,153.607
C07937=1083.018,121.440,432.577,174.677,21.658,153.607
C07938=1083.024,121.689,432.557,174.679,21.660,153.607
C07939=1083.029,121.938,432.537,174.681,21.663,153.607
C07940=1083.035,122.187,432.519,174.683,21.664,153.607
C07941=1083.039,122.437,432.499,174.685,21.666,153.607
C07942=1083.045,122.685,432.479,174.687,21.669,153.607
C07943=1083.051,122.935,432.459,174.688,21.670,153.607
C07944=1083.057,123.184,432.440,174.691,21.672,153.607
C07945=1083.063,123.434,432.421,174.693,21.674,153.607
C07946=1083.068,123.682,432.401,174.694,21.676,153.608
C07947=1083.074,123.931,432.382,174.697,21.679,153.608
C07948=1083.079,124.181,432.363,174.698,21.680,153.608
C07949=1083.085,124.430,432.343,174.700,21.682,153.608
C07950=1083.091,124.679,432.324,174.703,21.684,153.608
C07951=1083.097,124.928,432.304,174.704,21.686,153.608
C07952=1083.102,125.178,432.284,174.706,21.689,153.608
C07953=1083.108,125.427,432.265,174.709,21.690,153.608
C07954=1083.113,125.676,432.245,174.710,21.692,153.608
C07955=1083.119,125.925,432.225,174.713,21.694,153.608
C07956=1083.124,126.174,432.207,174.714,21.696,153.609
C07957=1083.130,126.423,432.187,174.716,21.698,153.609
C07958=1083.136,126.672,432.167,174.719,21.700,153.609
C07959=1083.142,126.922,432.148,174.720,21.702,153.609
C07960=1083.148,127.201,432.125,174.722,21.704,153.609
C07961=1083.154,127.481,432.103,174.725,21.706,153.609
C07962=1083.161,127.761,432.082,174.727,21.708,153.609
C07963=1083.168,128.040,432.059,174.729,21.711,153.609
C07964=1083.173,128.289,432.040,174.732,21.713,153.609
C07965=1083.179,128.537,432.020,174.733,21.714,153.609
C07966=1083.184,128.787,432.001,174.735,21.717,153.610
C07967=1083.190,129.036,431.981,174.738,21.719,153.610
C07968=1083.195,129.285,431.961,174.739,21.721,153.610
C07969=1083.201,129.534,431.941,174.742,21.722,153.610
C07970=1083.207,129.784,431.922,174.744,21.725,153.610
C07971=1083.213,130.032,431.902,174.745,21.726,153.610
C07972=1083.219,130.282,431.883,174.748,21.729,153.610
C07973=1083.224,130.531,431.862,174.749,21.730,153.610
C07974=1083.230,130.780,431.842,174.752,21.732,153.610
C07975=1083.236,131.029,431.823,174.754,21.734,153.610
C07976=1083.242,131.278,431.803,174.755,21.736,153.610
C07977=1083.247,131.528,431.784,174.758,21.738,153.610
C07978=1083.254,131.777,431.764,174.760,21.740,153.610
C07979=1083.259,132.026,431.743,174.761,21.742,153.611
C07980=1083.265,132.276,431.724,174.764,21.744,153.611
C07981=1083.271,132.524,431.704,174.766,21.746,153.611
C07982=1083.276,132.774,431.684,174.768,21.747,153.611
C07983=1083.282,133.023,431.664,174.770,21.750,153.611
C07984=1083.287,133.272,431.643,174.772,21.751,153.611
C07985=1083.293,133.522,431.624,174.774,21.753,153.611
C07986=1083.299,133.770,431.604,174.776,21.755,153.611
C07987=1083.304,134.019,431.584,174.778,21.758,153.611
C07988=1083.310,134.269,431.564,174.780,21.759,153.611
C07989=1083.315,134.518,431.544,174.782,21.761,153.612
C07990=1083.321,134.767,431.524,174.785,21.763,153.612
C07991=1083.327,135.016,431.504,174.786,21.765,153.612
C07992=1083.332,135.265,431.484,174.788,21.767,153.612
C07993=1083.338,135.514,431.464,174.791,21.769,153.612
C07994=1083.343,135.763,431.444,174.792,21.771,153.612
C07995=1083.349,136.012,431.424,174.795,21.773,153.612
C07996=1083.354,136.262,431.404,174.797,21.775,153.612
C07997=1083.360,136.511,431.384,174.799,21.776,153.612
C07998=1083.365,136.760,431.363,174.801,21.779,153.612
C07999=1083.371,137.009,431.343,174.803,21.781,153.612
C08000=1083.376,137.258,431.323,174.805,21.782,153.612
C08001=1083.382,137.507,431.304,174.807,21.784,153.612
C08002=1083.388,137.756,431.284,174.809,21.787,153.613
C08003=1083.393,138.005,431.263,174.811,21.788,153.613
C08004=1083.399,138.254,431.243,174.813,21.790,153.613
C08005=1083.405,138.503,431.222,174.815,21.792,153.613
C08006=1083.411,138.753,431.202,174.817,21.794,153.613
C08007=1083.416,139.002,431.182,174.819,21.796,153.613
C08008=1083.421,139.251,431.162,174.822,21.798,153.613
C08009=1083.427,139.500,431.142,174.824,21.800,153.613
C08010=1083.433,139.749,431.121,174.826,21.802,153.613
C08011=1083.439,139.998,431.101,174.828,21.803,153.613
C08012=1083.444,140.247,431.081,174.830,21.806,153.613
C08013=1083.450,140.496,431.061,174.832,21.807,153.613
C08014=1083.455,140.745,431.040,174.834,21.810,153.614
C08015=1083.461,140.995,431.019,174.836,21.811,153.614
C08016=1083.467,141.244,430.999,174.838,21.813,153.614
C08017=1083.472,141.493,430.979,174.840,21.815,153.614
C08018=1083.478,141.742,430.959,174.843,21.817,153.614
C08019=1083.484,141.991,430.938,174.845,21.819,153.614
C08020=1083.489,142.240,430.918,174.846,21.821,153.614
C08021=1083.495,142.489,430.898,174.849,21.823,153.614
C08022=1083.500,142.738,430.877,174.851,21.825,153.614
C08023=1083.505,142.987,430.857,174.853,21.826,153.614
C08024=1083.512,143.266,430.834,174.855,21.829,153.614
C08025=1083.519,143.546,430.811,174.857,21.831,153.614
C08026=1083.525,143.826,430.788,174.861,21.833,153.614
C08027=1083.531,144.105,430.765,174.863,21.835,153.614
C08028=1083.537,144.354,430.745,174.864,21.837,153.615
C08029=1083.542,144.603,430.724,174.867,21.839,153.615
C08030=1083.547,144.852,430.704,174.869,21.841,153.615
C08031=1083.553,145.102,430.683,174.871,21.843,153.615
C08032=1083.559,145.350,430.663,174.873,21.845,153.615
C08033=1083.565,145.600,430.641,174.875,21.847,153.615
C08034=1083.570,145.849,430.621,174.878,21.849,153.615
C08035=1083.576,146.098,430.601,174.879,21.850,153.615
C08036=1083.581,146.347,430.580,174.882,21.853,153.615
C08037=1083.587,146.597,430.559,174.884,21.854,153.615
C08038=1083.592,146.846,430.539,174.886,21.856,153.615
C08039=1083.599,147.094,430.518,174.888,21.858,153.615
C08040=1083.604,147.343,430.498,174.890,21.860,153.615
C08041=1083.609,147.592,430.477,174.893,21.862,153.615
C08042=1083.615,147.842,430.456,174.895,21.864,153.615
C08043=1083.621,148.091,430.436,174.896,21.866,153.616
C08044=1083.627,148.339,430.415,174.899,21.867,153.616
C08045=1083.632,148.588,430.394,174.901,21.869,153.616
C08046=1083.638,148.838,430.373,174.903,21.871,153.616
C08047=1083.643,149.087,430.352,174.905,21.873,153.616
C08048=1083.649,149.336,430.332,174.908,21.875,153.616
C08049=1083.655,149.585,430.312,174.910,21.877,153.616
C08050=1083.660,149.834,430.291,174.911,21.879,153.616
C08051=1083.666,150.083,430.269,174.914,21.880,153.616
C08052=1083.671,150.332,430.249,174.916,21.883,153.616
C08053=1083.676,150.581,430.228,174.919,21.885,153.616
C08054=1083.683,150.830,430.207,174.921,21.886,153.616
C08055=1083.688,151.080,430.186,174.922,21.888,153.616
C08056=1083.693,151.329,430.166,174.925,21.890,153.616
C08057=1083.699,151.577,430.144,174.927,21.892,153.616
C08058=1083.705,151.827,430.123,174.930,21.894,153.616
C08059=1083.710,152.075,430.102,174.931,21.896,153.616
C08060=1083.716,152.324,430.082,174.934,21.898,153.616
C08061=1083.722,152.574,430.061,174.936,21.900,153.616
C08062=1083.728,152.823,430.040,174.938,21.902,153.617
C08063=1083.733,153.072,430.019,174.940,21.903,153.617
C08064=1083.738,153.304,429.999,174.942,21.905,153.617
C08065=1083.743,153.538,429.980,174.945,21.907,153.617
C08066=1083.748,153.772,429.960,174.946,21.908,153.617
C08067=1083.754,154.004,429.940,174.948,21.911,153.617
C08068=1083.759,154.237,429.921,174.950,21.912,153.617
C08069=1083.764,154.470,429.901,174.952,21.914,153.617
C08070=1083.770,154.704,429.882,174.955,21.916,153.617
C08071=1083.775,154.936,429.862,174.957,21.917,153.617
C08072=1083.780,155.185,429.841,174.959,21.920,153.617
C08073=1083.786,155.434,429.820,174.961,21.921,153.617
C08074=1083.792,155.683,429.799,174.964,21.923,153.617
C08075=1083.797,155.932,429.777,174.965,21.925,153.617
C08076=1083.803,156.182,429.756,174.967,21.927,153.617
C08077=1083.808,156.431,429.735,174.970,21.929,153.617
C08078=1083.814,156.679,429.714,174.972,21.931,153.617
C08079=1083.819,156.929,429.693,174.975,21.932,153.617
C08080=1083.825,157.177,429.672,174.976,21.934,153.618
C08081=1083.830,157.426,429.651,174.979,21.936,153.618
C08082=1083.836,157.676,429.629,174.981,21.938,153.618
C08083=1083.842,157.924,429.608,174.984,21.940,153.618
C08084=1083.847,158.173,429.588,174.986,21.942,153.618
C08085=1083.853,158.423,429.565,174.987,21.944,153.618
C08086=1083.858,158.672,429.545,174.990,21.945,153.618
C08087=1083.864,158.921,429.523,174.992,21.947,153.618
C08088=1083.871,159.232,429.497,174.994,21.950,153.618
C08089=1083.878,159.543,429.470,174.998,21.952,153.618
C08090=1083.885,159.854,429.443,175.000,21.954,153.618
C08091=1083.892,160.165,429.417,175.003,21.957,153.618
C08092=1083.898,160.415,429.395,175.006,21.958,153.618
C08093=1083.903,160.664,429.374,175.008,21.960,153.618
C08094=1083.909,160.913,429.353,175.010,21.962,153.618
C08095=1083.915,161.161,429.332,175.012,21.964,153.618
C08096=1083.921,161.411,429.310,175.015,21.966,153.618
C08097=1083.925,161.660,429.289,175.017,21.968,153.618
C08098=1083.931,161.908,429.267,175.019,21.969,153.618
C08099=1083.937,162.158,429.246,175.022,21.972,153.618
C08100=1083.942,162.407,429.224,175.023,21.973,153.619
C08101=1083.947,162.656,429.203,175.026,21.975,153.619
C08102=1083.953,162.905,429.181,175.028,21.977,153.619
C08103=1083.958,163.154,429.160,175.030,21.979,153.619
C08104=1083.964,163.403,429.138,175.033,21.981,153.619
C08105=1083.969,163.652,429.116,175.035,21.983,153.619
C08106=1083.975,163.900,429.095,175.037,21.985,153.619
C08107=1083.980,164.150,429.073,175.039,21.987,153.619
C08108=1083.985,164.399,429.052,175.042,21.988,153.619
C08109=1083.991,164.648,429.030,175.044,21.991,153.619
C08110=1083.996,164.897,429.009,175.046,21.993,153.619
C08111=1084.001,165.146,428.987,175.049,21.994,153.619
C08112=1084.007,165.395,428.965,175.050,21.996,153.619
C08113=1084.012,165.644,428.944,175.053,21.998,153.619
C08114=1084.018,165.893,428.922,175.055,22.000,153.619
C08115=1084.023,166.142,428.900,175.057,22.002,153.619
C08116=1084.029,166.391,428.878,175.060,22.004,153.619
C08117=1084.035,166.639,428.857,175.062,22.006,153.619
C08118=1084.040,166.889,428.835,175.065,22.008,153.620
C08119=1084.046,167.137,428.814,175.066,22.009,153.620
C08120=1084.051,167.387,428.791,175.069,22.011,153.620
C08121=1084.057,167.635,428.770,175.071,22.013,153.620
C08122=1084.062,167.885,428.748,175.073,22.015,153.620
C08123=1084.068,168.133,428.727,175.076,22.017,153.620
C08124=1084.073,168.383,428.704,175.078,22.019,153.620
C08125=1084.078,168.632,428.683,175.081,22.021,153.620
C08126=1084.084,168.881,428.661,175.083,22.023,153.620
C08127=1084.089,169.130,428.639,175.084,22.025,153.620
C08128=1084.095,169.379,428.617,175.087,22.026,153.620
C08129=1084.100,169.628,428.596,175.089,22.028,153.620
C08130=1084.106,169.877,428.574,175.092,22.030,153.620
C08131=1084.111,170.125,428.551,175.094,22.032,153.620
C08132=1084.117,170.374,428.530,175.097,22.034,153.620
C08133=1084.122,170.623,428.508,175.099,22.036,153.620
C08134=1084.128,170.872,428.486,175.101,22.038,153.620
C08135=1084.133,171.121,428.464,175.103,22.039,153.620
C08136=1084.139,171.371,428.443,175.105,22.041,153.620
C08137=1084.145,171.619,428.420,175.108,22.043,153.620
C08138=1084.150,171.868,428.398,175.110,22.045,153.620
C08139=1084.156,172.117,428.376,175.113,22.047,153.620
C08140=1084.161,172.366,428.354,175.115,22.048,153.620
C08141=1084.167,172.615,428.333,175.118,22.051,153.620
C08142=1084.173,172.864,428.310,175.120,22.053,153.620
C08143=1084.178,173.113,428.289,175.122,22.054,153.620
C08144=1084.184,173.362,428.266,175.125,22.056,153.620
C08145=1084.189,173.611,428.244,175.126,22.058,153.621
C08146=1084.195,173.860,428.222,175.129,22.059,153.621
C08147=1084.201,174.109,428.200,175.131,22.061,153.621
C08148=1084.206,174.358,428.179,175.134,22.063,153.621
C08149=1084.212,174.607,428.156,175.136,22.065,153.621
C08150=1084.217,174.856,428.133,175.139,22.067,153.621
C08151=1084.223,175.105,428.112,175.141,22.069,153.621
C08152=1084.230,175.384,428.087,175.143,22.071,153.621
C08153=1084.235,175.662,428.062,175.146,22.073,153.621
C08154=1084.241,175.941,428.037,175.149,22.075,153.621
C08155=1084.248,176.221,428.012,175.152,22.077,153.621
C08156=1084.254,176.468,427.990,175.154,22.079,153.621
C08157=1084.259,176.718,427.968,175.157,22.081,153.621
C08158=1084.265,176.967,427.946,175.159,22.082,153.621
C08159=1084.271,177.215,427.924,175.161,22.084,153.621
C08160=1084.276,177.465,427.902,175.164,22.086,153.621
C08161=1084.282,177.714,427.879,175.166,22.088,153.621
C08162=1084.288,177.963,427.857,175.169,22.090,153.621
C08163=1084.293,178.211,427.834,175.170,22.091,153.621
C08164=1084.299,178.461,427.812,175.173,22.093,153.621
C08165=1084.305,178.709,427.790,175.175,22.095,153.621
C08166=1084.311,178.959,427.768,175.178,22.097,153.621
C08167=1084.316,179.207,427.745,175.180,22.098,153.621
C08168=1084.322,179.456,427.723,175.183,22.100,153.621
C08169=1084.328,179.705,427.701,175.185,22.102,153.621
C08170=1084.333,179.955,427.678,175.188,22.104,153.621
C08171=1084.338,180.203,427.656,175.190,22.106,153.621
C08172=1084.344,180.452,427.634,175.192,22.108,153.621
C08173=1084.350,180.701,427.611,175.195,22.109,153.621
C08174=1084.355,180.950,427.589,175.197,22.111,153.621
C08175=1084.362,181.199,427.567,175.200,22.113,153.621
C08176=1084.367,181.447,427.544,175.202,22.115,153.621
C08177=1084.372,181.697,427.522,175.205,22.117,153.621
C08178=1084.378,181.946,427.499,175.207,22.119,153.621
C08179=1084.384,182.195,427.477,175.210,22.120,153.621
C08180=1084.390,182.444,427.454,175.212,22.122,153.621
C08181=1084.396,182.693,427.431,175.215,22.123,153.621
C08182=1084.401,182.941,427.409,175.217,22.125,153.621
C08183=1084.407,183.190,427.387,175.220,22.127,153.621
C08184=1084.413,183.439,427.364,175.222,22.129,153.621
C08185=1084.418,183.688,427.342,175.224,22.130,153.621
C08186=1084.424,183.937,427.319,175.226,22.132,153.621
C08187=1084.430,184.186,427.297,175.229,22.134,153.621
C08188=1084.436,184.435,427.274,175.231,22.136,153.621
C08189=1084.441,184.684,427.252,175.233,22.138,153.621
C08190=1084.447,184.933,427.229,175.236,22.139,153.621
C08191=1084.452,185.181,427.206,175.239,22.141,153.621
C08192=1084.458,185.430,427.183,175.241,22.143,153.621
C08193=1084.464,185.680,427.161,175.243,22.145,153.621
C08194=1084.469,185.928,427.138,175.246,22.147,153.621
C08195=1084.474,186.177,427.115,175.248,22.149,153.621
C08196=1084.480,186.426,427.092,175.251,22.150,153.621
C08197=1084.486,186.675,427.069,175.253,22.152,153.621
C08198=1084.491,186.924,427.047,175.256,22.154,153.621
C08199=1084.496,187.173,427.024,175.258,22.156,153.621
C08200=1084.502,187.422,427.001,175.260,22.158,153.621
C08201=1084.507,187.671,426.978,175.263,22.160,153.622
C08202=1084.513,187.919,426.955,175.265,22.162,153.622
C08203=1084.519,188.168,426.932,175.268,22.164,153.622
C08204=1084.524,188.417,426.910,175.270,22.166,153.622
C08205=1084.529,188.666,426.886,175.273,22.167,153.622
C08206=1084.535,188.915,426.863,175.275,22.169,153.622
C08207=1084.540,189.164,426.841,175.277,22.171,153.622
C08208=1084.546,189.413,426.818,175.280,22.173,153.622
C08209=1084.551,189.662,426.795,175.283,22.175,153.622
C08210=1084.557,189.911,426.772,175.286,22.177,153.622
C08211=1084.562,190.159,426.749,175.288,22.179,153.622
C08212=1084.567,190.408,426.726,175.291,22.181,153.622
C08213=1084.573,190.657,426.703,175.293,22.182,153.622
C08214=1084.579,190.906,426.680,175.296,22.184,153.622
C08215=1084.584,191.155,426.657,175.298,22.186,153.622
C08216=1084.590,191.433,426.631,175.300,22.188,153.622
C08217=1084.597,191.712,426.604,175.303,22.190,153.622
C08218=1084.603,191.990,426.580,175.306,22.193,153.622
C08219=1084.609,192.268,426.553,175.309,22.194,153.622
C08220=1084.615,192.517,426.531,175.311,22.196,153.622
C08221=1084.620,192.766,426.507,175.313,22.198,153.622
C08222=1084.625,193.015,426.484,175.316,22.200,153.622
C08223=1084.631,193.264,426.461,175.318,22.202,153.622
C08224=1084.637,193.513,426.438,175.322,22.204,153.622
C08225=1084.642,193.762,426.414,175.324,22.206,153.622
C08226=1084.648,194.011,426.391,175.327,22.208,153.622
C08227=1084.654,194.259,426.368,175.329,22.209,153.622
C08228=1084.659,194.508,426.345,175.332,22.211,153.622
C08229=1084.664,194.758,426.322,175.334,22.213,153.622
C08230=1084.670,195.006,426.299,175.336,22.215,153.622
C08231=1084.676,195.255,426.275,175.339,22.217,153.622
C08232=1084.682,195.504,426.252,175.341,22.218,153.622
C08233=1084.687,195.753,426.228,175.344,22.220,153.622
C08234=1084.693,196.002,426.205,175.346,22.222,153.622
C08235=1084.699,196.250,426.182,175.349,22.223,153.622
C08236=1084.704,196.499,426.158,175.351,22.225,153.622
C08237=1084.709,196.748,426.135,175.354,22.227,153.622
C08238=1084.715,196.997,426.112,175.356,22.229,153.622
C08239=1084.720,197.246,426.088,175.360,22.231,153.622
C08240=1084.726,197.494,426.065,175.362,22.233,153.622
C08241=1084.732,197.743,426.042,175.365,22.235,153.622
C08242=1084.738,197.992,426.019,175.367,22.237,153.622
C08243=1084.743,198.241,425.995,175.369,22.238,153.622
C08244=1084.749,198.490,425.972,175.372,22.240,153.622
C08245=1084.755,198.739,425.948,175.374,22.242,153.622
C08246=1084.760,198.988,425.925,175.377,22.244,153.622
C08247=1084.766,199.237,425.902,175.379,22.246,153.622
C08248=1084.772,199.485,425.878,175.382,22.247,153.622
C08249=1084.777,199.734,425.854,175.384,22.249,153.622
C08250=1084.783,199.983,425.831,175.388,22.251,153.622
C08251=1084.788,200.232,425.807,175.390,22.253,153.622
C08252=1084.794,200.481,425.784,175.393,22.255,153.622
C08253=1084.800,200.730,425.760,175.395,22.257,153.622
C08254=1084.805,200.979,425.737,175.398,22.258,153.622
C08255=1084.811,201.227,425.713,175.400,22.260,153.622
C08256=1084.817,201.476,425.690,175.403,22.262,153.622
C08257=1084.822,201.725,425.666,175.405,22.263,153.622
C08258=1084.828,201.974,425.643,175.408,22.265,153.622
C08259=1084.833,202.222,425.619,175.411,22.267,153.622
C08260=1084.840,202.472,425.595,175.413,22.269,153.622
C08261=1084.846,202.720,425.572,175.416,22.271,153.622
C08262=1084.851,202.969,425.548,175.418,22.273,153.622
C08263=1084.856,203.218,425.524,175.421,22.275,153.622
C08264=1084.862,203.466,425.500,175.423,22.277,153.622
C08265=1084.867,203.715,425.477,175.426,22.278,153.622
C08266=1084.873,203.964,425.453,175.428,22.280,153.622
C08267=1084.878,204.213,425.429,175.432,22.283,153.622
C08268=1084.884,204.462,425.405,175.434,22.284,153.622
C08269=1084.890,204.710,425.381,175.436,22.286,153.622
C08270=1084.895,204.960,425.358,175.439,22.288,153.622
C08271=1084.901,205.208,425.334,175.441,22.290,153.622
C08272=1084.906,205.456,425.310,175.444,22.292,153.622
C08273=1084.911,205.706,425.286,175.447,22.294,153.622
C08274=1084.918,205.955,425.262,175.450,22.296,153.622
C08275=1084.923,206.203,425.238,175.452,22.298,153.622
C08276=1084.928,206.452,425.214,175.455,22.299,153.622
C08277=1084.934,206.701,425.191,175.457,22.301,153.622
C08278=1084.940,206.949,425.166,175.459,22.303,153.623
C08279=1084.946,207.199,425.142,175.462,22.305,153.623
C08280=1084.969,208.227,425.044,175.546,22.349,153.619
C08281=1084.978,208.616,425.005,175.551,22.354,153.620
C08282=1084.987,209.005,424.967,175.554,22.358,153.620
C08283=1084.995,209.395,424.929,175.558,22.362,153.621
C08284=1085.004,209.785,424.890,175.562,22.366,153.621
C08285=1085.009,210.033,424.866,175.565,22.369,153.621
C08286=1085.015,210.281,424.841,175.567,22.372,153.621
C08287=1085.021,210.531,424.816,175.570,22.375,153.622
C08288=1085.026,210.779,424.792,175.572,22.377,153.622
C08289=1085.032,211.029,424.768,175.574,22.380,153.622
C08290=1085.037,211.277,424.743,175.577,22.383,153.622
C08291=1085.044,211.526,424.718,175.579,22.386,153.622
C08292=1085.049,211.774,424.694,175.581,22.389,153.623
C08293=1085.054,212.023,424.670,175.585,22.391,153.623
C08294=1085.060,212.272,424.644,175.587,22.394,153.623
C08295=1085.066,212.520,424.620,175.590,22.397,153.623
C08296=1085.072,212.770,424.595,175.592,22.400,153.624
C08297=1085.077,213.018,424.571,175.594,22.402,153.624
C08298=1085.083,213.267,424.546,175.597,22.405,153.624
C08299=1085.088,213.515,424.521,175.599,22.408,153.624
C08300=1085.094,213.765,424.497,175.602,22.411,153.625
C08301=1085.100,214.013,424.472,175.605,22.414,153.625
C08302=1085.106,214.262,424.447,175.607,22.416,153.625
C08303=1085.111,214.510,424.422,175.610,22.420,153.625
C08304=1085.116,214.759,424.397,175.612,22.422,153.625
C08305=1085.122,215.008,424.373,175.615,22.425,153.626
C08306=1085.127,215.256,424.348,175.617,22.428,153.626
C08307=1085.133,215.505,424.323,175.620,22.431,153.626
C08308=1085.139,215.753,424.298,175.622,22.434,153.626
C08309=1085.145,216.003,424.274,175.625,22.436,153.627
C08310=1085.150,216.252,424.248,175.627,22.439,153.627
C08311=1085.156,216.500,424.223,175.630,22.442,153.627
C08312=1085.162,216.749,424.198,175.633,22.445,153.627
C08313=1085.167,216.997,424.174,175.635,22.448,153.627
C08314=1085.173,217.246,424.148,175.637,22.450,153.628
C08315=1085.178,217.495,424.124,175.640,22.453,153.628
C08316=1085.184,217.744,424.098,175.642,22.456,153.628
C08317=1085.189,217.992,424.074,175.645,22.459,153.628
C08318=1085.196,218.241,424.049,175.647,22.462,153.629
C08319=1085.200,218.489,424.023,175.650,22.465,153.629
C08320=1085.206,218.738,423.998,175.653,22.467,153.629
C08321=1085.213,218.987,423.973,175.655,22.470,153.629
C08322=1085.218,219.236,423.949,175.658,22.473,153.629
C08323=1085.223,219.485,423.923,175.660,22.475,153.630
C08324=1085.229,219.733,423.898,175.663,22.479,153.630
C08325=1085.235,219.982,423.873,175.665,22.481,153.630
C08326=1085.241,220.231,423.848,175.668,22.484,153.630
C08327=1085.246,220.479,423.822,175.671,22.487,153.631
C08328=1085.252,220.728,423.798,175.674,22.490,153.631
C08329=1085.258,220.977,423.773,175.676,22.493,153.631
C08330=1085.264,221.225,423.748,175.678,22.495,153.631
C08331=1085.269,221.474,423.722,175.681,22.498,153.632
C08332=1085.275,221.723,423.697,175.683,22.501,153.632
C08333=1085.284,222.116,423.657,175.688,22.505,153.632
C08334=1085.292,222.509,423.617,175.691,22.510,153.633
C08335=1085.301,222.902,423.577,175.696,22.514,153.633
C08336=1085.310,223.295,423.536,175.700,22.519,153.633
C08337=1085.316,223.545,423.512,175.702,22.522,153.634
C08338=1085.321,223.794,423.486,175.705,22.524,153.634
C08339=1085.327,224.042,423.461,175.708,22.527,153.634
C08340=1085.332,224.291,423.435,175.710,22.530,153.634
C08341=1085.339,224.539,423.410,175.713,22.533,153.634
C08342=1085.344,224.788,423.384,175.715,22.536,153.635
C08343=1085.350,225.036,423.359,175.718,22.539,153.635
C08344=1085.355,225.285,423.333,175.720,22.541,153.635
C08345=1085.361,225.533,423.308,175.723,22.544,153.635
C08346=1085.366,225.782,423.282,175.725,22.547,153.636
C08347=1085.372,226.031,423.257,175.728,22.550,153.636
C08348=1085.378,226.280,423.231,175.731,22.553,153.636
C08349=1085.384,226.528,423.206,175.733,22.556,153.636
C08350=1085.389,226.777,423.180,175.736,22.559,153.637
C08351=1085.394,227.026,423.154,175.738,22.561,153.637
C08352=1085.400,227.274,423.129,175.741,22.564,153.637
C08353=1085.406,227.523,423.103,175.743,22.567,153.637
C08354=1085.412,227.771,423.078,175.746,22.570,153.637
C08355=1085.417,228.020,423.052,175.749,22.572,153.638
C08356=1085.423,228.269,423.026,175.752,22.576,153.638
C08357=1085.428,228.517,423.001,175.754,22.578,153.638
C08358=1085.435,228.766,422.975,175.757,22.581,153.638
C08359=1085.440,229.015,422.949,175.759,22.584,153.639
C08360=1085.445,229.264,422.924,175.762,22.587,153.639
C08361=1085.452,229.513,422.898,175.764,22.590,153.639
C08362=1085.457,229.760,422.872,175.767,22.593,153.639
C08363=1085.463,230.009,422.847,175.770,22.595,153.639
C08364=1085.469,230.258,422.821,175.773,22.598,153.640
C08365=1085.474,230.507,422.795,175.775,22.601,153.640
C08366=1085.480,230.756,422.769,175.778,22.604,153.640
C08367=1085.485,231.003,422.743,175.780,22.607,153.640
C08368=1085.491,231.252,422.717,175.783,22.609,153.641
C08369=1085.496,231.501,422.691,175.785,22.612,153.641
C08370=1085.502,231.750,422.666,175.788,22.615,153.641
C08371=1085.508,231.998,422.639,175.791,22.618,153.641
C08372=1085.514,232.247,422.613,175.794,22.621,153.642
C08373=1085.519,232.496,422.588,175.796,22.624,153.642
C08374=1085.525,232.744,422.562,175.799,22.627,153.642
C08375=1085.531,232.993,422.536,175.802,22.630,153.642
C08376=1085.536,233.242,422.510,175.804,22.633,153.643
C08377=1085.542,233.490,422.483,175.807,22.635,153.643
C08378=1085.547,233.739,422.457,175.809,22.638,153.643
C08379=1085.554,233.988,422.432,175.812,22.641,153.643
C08380=1085.559,234.235,422.406,175.814,22.644,153.644
C08381=1085.564,234.484,422.380,175.817,22.647,153.644
C08382=1085.570,234.733,422.354,175.820,22.650,153.644
C08383=1085.575,234.982,422.327,175.823,22.653,153.644
C08384=1085.581,235.230,422.301,175.825,22.655,153.644
C08385=1085.589,235.609,422.261,175.829,22.660,153.645
C08386=1085.598,235.988,422.221,175.833,22.664,153.645
C08387=1085.607,236.366,422.181,175.838,22.669,153.646
C08388=1085.615,236.745,422.142,175.841,22.673,153.646
C08389=1085.621,236.994,422.115,175.843,22.676,153.646
C08390=1085.626,237.242,422.088,175.847,22.679,153.646
C08391=1085.632,237.491,422.063,175.850,22.682,153.647
C08392=1085.638,237.739,422.036,175.852,22.685,153.647
C08393=1085.643,237.988,422.010,175.855,22.687,153.647
C08394=1085.649,238.237,421.983,175.857,22.690,153.647
C08395=1085.654,238.486,421.957,175.860,22.693,153.648
C08396=1085.661,238.734,421.931,175.862,22.696,153.648
C08397=1085.667,238.982,421.905,175.865,22.699,153.648
C08398=1085.672,239.231,421.879,175.868,22.702,153.648
C08399=1085.678,239.479,421.852,175.871,22.705,153.649
C08400=1085.684,239.728,421.825,175.874,22.708,153.649
C08401=1085.689,239.977,421.799,175.876,22.711,153.649
C08402=1085.695,240.225,421.773,175.879,22.713,153.649
C08403=1085.701,240.473,421.746,175.881,22.716,153.650
C08404=1085.706,240.722,421.719,175.884,22.719,153.650
C08405=1085.711,240.971,421.693,175.887,22.722,153.650
C08406=1085.717,241.219,421.666,175.889,22.725,153.650
C08407=1085.723,241.468,421.640,175.892,22.728,153.650
C08408=1085.728,241.716,421.613,175.895,22.730,153.651
C08409=1085.734,241.965,421.587,175.898,22.734,153.651
C08410=1085.740,242.214,421.560,175.900,22.736,153.651
C08411=1085.746,242.462,421.534,175.903,22.739,153.651
C08412=1085.751,242.710,421.507,175.906,22.742,153.652
C08413=1085.757,242.965,421.480,175.908,22.745,153.652
C08414=1085.763,243.220,421.452,175.911,22.748,153.652
C08415=1085.769,243.474,421.425,175.914,22.751,153.652
C08416=1085.775,243.729,421.398,175.916,22.754,153.653
C08417=1085.780,243.978,421.371,175.919,22.757,153.653
C08418=1085.786,244.226,421.344,175.922,22.760,153.653
C08419=1085.791,244.474,421.318,175.924,22.763,153.653
C08420=1085.797,244.723,421.291,175.928,22.766,153.654
C08421=1085.802,244.971,421.264,175.930,22.769,153.654
C08422=1085.808,245.220,421.237,175.933,22.772,153.654
C08423=1085.814,245.468,421.211,175.936,22.775,153.654
C08424=1085.820,245.716,421.184,175.938,22.777,153.655
C08425=1085.825,245.965,421.157,175.941,22.781,153.655
C08426=1085.831,246.214,421.130,175.943,22.783,153.655
C08427=1085.837,246.462,421.103,175.946,22.787,153.655
C08428=1085.842,246.711,421.076,175.949,22.789,153.656
C08429=1085.848,246.959,421.049,175.951,22.792,153.656
C08430=1085.853,247.208,421.022,175.954,22.795,153.656
C08431=1085.858,247.457,420.995,175.957,22.798,153.656
C08432=1085.864,247.705,420.969,175.960,22.801,153.657
C08433=1085.870,247.953,420.942,175.963,22.804,153.657
C08434=1085.875,248.202,420.915,175.965,22.807,153.657
C08435=1085.882,248.450,420.887,175.968,22.810,153.657
C08436=1085.887,248.699,420.860,175.971,22.813,153.658
C08437=1085.895,249.077,420.819,175.975,22.817,153.658
C08438=1085.904,249.454,420.777,175.979,22.822,153.659
C08439=1085.912,249.832,420.736,175.983,22.827,153.659
C08440=1085.920,250.210,420.695,175.987,22.831,153.659
C08441=1085.926,250.459,420.668,175.990,22.834,153.660
C08442=1085.932,250.708,420.641,175.993,22.837,153.660
C08443=1085.937,250.956,420.614,175.996,22.840,153.660
C08444=1085.943,251.204,420.586,175.998,22.843,153.660
C08445=1085.948,251.453,420.559,176.001,22.846,153.661
C08446=1085.954,251.702,420.532,176.004,22.849,153.661
C08447=1085.960,251.950,420.504,176.006,22.852,153.661
C08448=1085.965,252.199,420.477,176.009,22.855,153.661
C08449=1085.970,252.447,420.450,176.011,22.858,153.662
C08450=1085.976,252.695,420.422,176.014,22.861,153.662
C08451=1085.982,252.944,420.395,176.017,22.864,153.662
C08452=1085.988,253.192,420.367,176.020,22.866,153.662
C08453=1085.993,253.440,420.341,176.023,22.870,153.663
C08454=1085.998,253.689,420.313,176.026,22.873,153.663
C08455=1086.005,253.938,420.286,176.028,22.876,153.663
C08456=1086.010,254.186,420.258,176.031,22.879,153.664
C08457=1086.015,254.434,420.230,176.034,22.882,153.664
C08458=1086.021,254.683,420.204,176.036,22.884,153.664
C08459=1086.027,254.931,420.175,176.039,22.888,153.664
C08460=1086.033,255.180,420.149,176.042,22.891,153.665
C08461=1086.038,255.428,420.121,176.044,22.894,153.665
C08462=1086.044,255.677,420.093,176.047,22.897,153.665
C08463=1086.050,255.925,420.066,176.050,22.900,153.665
C08464=1086.055,256.174,420.039,176.053,22.902,153.666
C08465=1086.062,256.422,420.011,176.056,22.905,153.666
C08466=1086.067,256.671,419.984,176.059,22.909,153.666
C08467=1086.072,256.919,419.956,176.062,22.912,153.666
C08468=1086.079,257.167,419.928,176.064,22.915,153.667
C08469=1086.084,257.416,419.901,176.067,22.917,153.667
C08470=1086.089,257.664,419.873,176.070,22.921,153.667
C08471=1086.096,257.912,419.845,176.072,22.923,153.667
C08472=1086.101,258.161,419.818,176.075,22.927,153.668
C08473=1086.106,258.409,419.790,176.078,22.930,153.668
C08474=1086.113,258.658,419.762,176.080,22.932,153.668
C08475=1086.118,258.906,419.735,176.083,22.935,153.668
C08476=1086.124,259.155,419.707,176.086,22.938,153.669
C08477=1086.130,259.403,419.679,176.089,22.941,153.669
C08478=1086.135,259.651,419.651,176.092,22.944,153.669
C08479=1086.141,259.900,419.624,176.095,22.947,153.669
C08480=1086.147,260.148,419.596,176.098,22.950,153.670
C08481=1086.153,260.397,419.568,176.100,22.953,153.670
C08482=1086.158,260.645,419.540,176.103,22.956,153.670
C08483=1086.165,260.893,419.512,176.106,22.960,153.670
C08484=1086.170,261.142,419.485,176.108,22.962,153.671
C08485=1086.175,261.390,419.457,176.111,22.965,153.671
C08486=1086.181,261.639,419.429,176.114,22.968,153.671
C08487=1086.187,261.886,419.401,176.116,22.971,153.671
C08488=1086.193,262.135,419.373,176.120,22.974,153.672
C08489=1086.202,262.511,419.331,176.124,22.979,153.672
C08490=1086.211,262.885,419.289,176.128,22.983,153.672
C08491=1086.219,263.261,419.247,176.133,22.987,153.673
C08492=1086.229,263.636,419.204,176.137,22.992,153.673
C08493=1086.234,263.884,419.176,176.139,22.995,153.673
C08494=1086.240,264.132,419.148,176.142,22.998,153.674
C08495=1086.245,264.380,419.120,176.145,23.001,153.674
C08496=1086.251,264.629,419.092,176.148,23.004,153.674
C08497=1086.257,264.877,419.064,176.150,23.007,153.675
C08498=1086.262,265.126,419.035,176.154,23.010,153.675
C08499=1086.268,265.374,419.008,176.157,23.013,153.675
C08500=1086.274,265.623,418.979,176.160,23.017,153.675
C08501=1086.279,265.871,418.951,176.162,23.019,153.676
C08502=1086.285,266.119,418.922,176.165,23.022,153.676
C08503=1086.291,266.367,418.894,176.168,23.025,153.676
C08504=1086.297,266.616,418.866,176.170,23.028,153.676
C08505=1086.302,266.864,418.838,176.173,23.031,153.677
C08506=1086.308,267.113,418.810,176.176,23.034,153.677
C08507=1086.313,267.361,418.782,176.179,23.038,153.677
C08508=1086.319,267.609,418.753,176.181,23.040,153.678
C08509=1086.325,267.857,418.725,176.184,23.044,153.678
C08510=1086.331,268.106,418.696,176.187,23.047,153.678
C08511=1086.337,268.354,418.668,176.190,23.050,153.678
C08512=1086.342,268.602,418.640,176.193,23.053,153.679
C08513=1086.348,268.850,418.611,176.196,23.056,153.679
C08514=1086.354,269.099,418.583,176.199,23.059,153.679
C08515=1086.360,269.347,418.555,176.202,23.062,153.680
C08516=1086.366,269.595,418.526,176.205,23.065,153.680
C08517=1086.370,269.844,418.497,176.207,23.068,153.680
C08518=1086.376,270.093,418.469,176.210,23.071,153.680
C08519=1086.382,270.340,418.440,176.213,23.075,153.681
C08520=1086.388,270.589,418.412,176.216,23.078,153.681
C08521=1086.393,270.837,418.384,176.218,23.081,153.681
C08522=1086.399,271.085,418.354,176.221,23.084,153.682
C08523=1086.405,271.334,418.326,176.224,23.087,153.682
C08524=1086.410,271.581,418.297,176.227,23.090,153.682
C08525=1086.416,271.830,418.269,176.230,23.093,153.682
C08526=1086.422,272.079,418.241,176.232,23.096,153.683
C08527=1086.427,272.327,418.211,176.235,23.099,153.683
C08528=1086.433,272.575,418.183,176.238,23.102,153.683
C08529=1086.439,272.823,418.154,176.241,23.106,153.684
C08530=1086.445,273.072,418.126,176.244,23.108,153.684
C08531=1086.450,273.320,418.096,176.247,23.112,153.684
C08532=1086.456,273.568,418.068,176.250,23.115,153.684
C08533=1086.462,273.816,418.039,176.253,23.118,153.685
C08534=1086.468,274.064,418.010,176.256,23.121,153.685
C08535=1086.473,274.313,417.982,176.258,23.124,153.685
C08536=1086.479,274.561,417.953,176.261,23.128,153.686
C08537=1086.484,274.810,417.924,176.264,23.131,153.686
C08538=1086.490,275.057,417.895,176.267,23.134,153.686
C08539=1086.496,275.305,417.866,176.270,23.137,153.687
C08540=1086.501,275.554,417.837,176.272,23.140,153.687
C08541=1086.510,275.932,417.793,176.276,23.145,153.687
C08542=1086.519,276.311,417.749,176.281,23.150,153.688
C08543=1086.528,276.688,417.705,176.286,23.154,153.688
C08544=1086.536,277.066,417.662,176.290,23.159,153.689
C08545=1086.542,277.314,417.632,176.292,23.162,153.689
C08546=1086.548,277.562,417.603,176.295,23.165,153.689
C08547=1086.553,277.811,417.573,176.298,23.169,153.689
C08548=1086.559,278.059,417.545,176.301,23.172,153.690
C08549=1086.564,278.307,417.516,176.304,23.175,153.690
C08550=1086.570,278.556,417.487,176.307,23.179,153.690
C08551=1086.576,278.804,417.457,176.309,23.181,153.691
C08552=1086.582,279.051,417.428,176.312,23.184,153.691
C08553=1086.588,279.300,417.399,176.316,23.188,153.691
C08554=1086.593,279.548,417.370,176.319,23.191,153.692
C08555=1086.599,279.797,417.341,176.321,23.195,153.692
C08556=1086.605,280.045,417.312,176.324,23.198,153.692
C08557=1086.610,280.293,417.282,176.327,23.200,153.693
C08558=1086.616,280.541,417.253,176.330,23.204,153.693
C08559=1086.621,280.789,417.224,176.333,23.207,153.693
C08560=1086.628,281.038,417.195,176.336,23.210,153.693
C08561=1086.633,281.286,417.165,176.339,23.214,153.694
C08562=1086.639,281.533,417.136,176.342,23.217,153.694
C08563=1086.644,281.782,417.107,176.344,23.220,153.694
C08564=1086.650,282.030,417.077,176.347,23.223,153.695
C08565=1086.656,282.279,417.048,176.350,23.226,153.695
C08566=1086.662,282.527,417.018,176.353,23.230,153.695
C08567=1086.667,282.775,416.989,176.356,23.233,153.696
C08568=1086.673,283.023,416.960,176.359,23.236,153.696
C08569=1086.678,283.271,416.930,176.362,23.240,153.696
C08570=1086.684,283.519,416.900,176.364,23.242,153.697
C08571=1086.690,283.768,416.870,176.367,23.245,153.697
C08572=1086.696,284.016,416.841,176.370,23.249,153.697
C08573=1086.701,284.264,416.812,176.373,23.252,153.698
C08574=1086.706,284.512,416.783,176.376,23.255,153.698
C08575=1086.713,284.760,416.753,176.379,23.259,153.698
C08576=1086.718,285.008,416.724,176.382,23.262,153.699
C08577=1086.724,285.256,416.693,176.385,23.265,153.699
C08578=1086.729,285.505,416.664,176.387,23.268,153.699
C08579=1086.736,285.753,416.635,176.390,23.272,153.700
C08580=1086.741,286.001,416.605,176.393,23.275,153.700
C08581=1086.747,286.249,416.575,176.396,23.278,153.700
C08582=1086.753,286.498,416.545,176.399,23.282,153.701
C08583=1086.759,286.746,416.516,176.402,23.285,153.701
C08584=1086.765,286.993,416.486,176.405,23.288,153.701
C08585=1086.769,287.241,416.457,176.408,23.292,153.702
C08586=1086.775,287.490,416.427,176.411,23.295,153.702
C08587=1086.781,287.737,416.397,176.413,23.298,153.702
C08588=1086.787,287.986,416.367,176.416,23.301,153.703
C08589=1086.793,288.234,416.338,176.419,23.305,153.703
C08590=1086.798,288.482,416.308,176.422,23.308,153.703
C08591=1086.804,288.730,416.278,176.425,23.311,153.703
C08592=1086.810,288.978,416.248,176.428,23.315,153.704
C08593=1086.819,289.366,416.201,176.433,23.320,153.704
C08594=1086.828,289.753,416.154,176.437,23.325,153.705
C08595=1086.837,290.141,416.108,176.441,23.330,153.706
C08596=1086.846,290.529,416.060,176.446,23.335,153.706
C08597=1086.852,290.777,416.031,176.449,23.338,153.706
C08598=1086.857,291.025,416.000,176.452,23.342,153.707
C08599=1086.863,291.273,415.971,176.455,23.345,153.707
C08600=1086.869,291.521,415.941,176.458,23.349,153.707
C08601=1086.875,291.769,415.910,176.461,23.352,153.708
C08602=1086.880,292.018,415.881,176.464,23.355,153.708
C08603=1086.886,292.265,415.850,176.467,23.359,153.708
C08604=1086.891,292.514,415.821,176.470,23.362,153.709
C08605=1086.897,292.762,415.790,176.473,23.365,153.709
C08606=1086.903,293.009,415.760,176.476,23.369,153.710
C08607=1086.909,293.258,415.730,176.479,23.372,153.710
C08608=1086.914,293.506,415.700,176.482,23.376,153.710
C08609=1086.920,293.754,415.670,176.484,23.379,153.711
C08610=1086.926,294.001,415.639,176.487,23.382,153.711
C08611=1086.931,294.250,415.610,176.490,23.385,153.711
C08612=1086.937,294.498,415.579,176.493,23.389,153.712
C08613=1086.943,294.745,415.549,176.496,23.392,153.712
C08614=1086.949,294.993,415.518,176.499,23.396,153.712
C08615=1086.955,295.242,415.487,176.502,23.399,153.713
C08616=1086.960,295.491,415.458,176.505,23.403,153.713
C08617=1086.966,295.738,415.427,176.508,23.406,153.713
C08618=1086.972,295.986,415.397,176.511,23.409,153.714
C08619=1086.978,296.234,415.366,176.514,23.413,153.714
C08620=1086.983,296.482,415.336,176.516,23.416,153.714
C08621=1086.989,296.730,415.306,176.520,23.419,153.715
C08622=1086.994,296.978,415.275,176.522,23.423,153.715
C08623=1087.000,297.227,415.245,176.525,23.427,153.716
C08624=1087.006,297.475,415.214,176.528,23.430,153.716
C08625=1087.012,297.723,415.184,176.531,23.433,153.716
C08626=1087.018,297.970,415.154,176.534,23.437,153.717
C08627=1087.023,298.219,415.123,176.537,23.440,153.717
C08628=1087.029,298.466,415.092,176.540,23.444,153.717
C08629=1087.034,298.714,415.062,176.543,23.447,153.718
C08630=1087.040,298.963,415.031,176.546,23.451,153.718
C08631=1087.046,299.211,415.000,176.549,23.454,153.719
C08632=1087.051,299.459,414.970,176.552,23.458,153.719
C08633=1087.057,299.706,414.938,176.555,23.461,153.719
C08634=1087.062,299.954,414.908,176.558,23.465,153.720
C08635=1087.068,300.202,414.877,176.561,23.468,153.720
C08636=1087.073,300.450,414.846,176.564,23.472,153.721
C08637=1087.080,300.699,414.815,176.567,23.476,153.721
C08638=1087.085,300.947,414.785,176.569,23.479,153.721
C08639=1087.091,301.195,414.754,176.572,23.483,153.722
C08640=1087.096,301.443,414.724,176.575,23.486,153.722
C08641=1087.102,301.690,414.692,176.578,23.490,153.722
C08642=1087.108,301.938,414.662,176.581,23.493,153.723
C08643=1087.113,302.187,414.631,176.584,23.497,153.723
C08644=1087.119,302.435,414.600,176.587,23.500,153.724
C08645=1087.128,302.836,414.550,176.591,23.506,153.724
C08646=1087.137,303.237,414.499,176.597,23.512,153.725
C08647=1087.146,303.639,414.450,176.601,23.517,153.726
C08648=1087.155,304.041,414.399,176.606,23.524,153.726
C08649=1087.161,304.289,414.369,176.609,23.527,153.727
C08650=1087.167,304.536,414.337,176.612,23.530,153.727
C08651=1087.173,304.785,414.306,176.615,23.534,153.727
C08652=1087.178,305.032,414.275,176.618,23.538,153.728
C08653=1087.184,305.280,414.244,176.621,23.541,153.728
C08654=1087.190,305.528,414.212,176.624,23.545,153.729
C08655=1087.195,305.777,414.181,176.627,23.548,153.729
C08656=1087.201,306.024,414.151,176.630,23.552,153.730
C08657=1087.207,306.273,414.119,176.633,23.555,153.730
C08658=1087.213,306.520,414.089,176.636,23.559,153.730
C08659=1087.218,306.768,414.057,176.638,23.562,153.731
C08660=1087.225,307.016,414.026,176.641,23.566,153.731
C08661=1087.230,307.264,413.995,176.645,23.570,153.732
C08662=1087.236,307.511,413.963,176.648,23.574,153.732
C08663=1087.242,307.760,413.932,176.651,23.577,153.732
C08664=1087.247,308.008,413.901,176.654,23.581,153.733
C08665=1087.254,308.256,413.870,176.657,23.585,153.733
C08666=1087.259,308.504,413.838,176.660,23.588,153.734
C08667=1087.264,308.752,413.807,176.663,23.592,153.734
C08668=1087.271,309.000,413.776,176.666,23.595,153.734
C08669=1087.276,309.247,413.744,176.668,23.599,153.735
C08670=1087.282,309.496,413.713,176.672,23.602,153.735
C08671=1087.288,309.743,413.682,176.674,23.606,153.736
C08672=1087.294,309.991,413.650,176.677,23.609,153.736
C08673=1087.300,310.239,413.618,176.680,23.613,153.736
C08674=1087.306,310.487,413.587,176.683,23.617,153.737
C08675=1087.311,310.735,413.556,176.687,23.621,153.737
C08676=1087.317,310.983,413.524,176.690,23.624,153.738
C08677=1087.323,311.231,413.493,176.693,23.628,153.738
C08678=1087.329,311.479,413.461,176.696,23.632,153.739
C08679=1087.335,311.727,413.430,176.699,23.635,153.739
C08680=1087.341,311.975,413.398,176.702,23.639,153.739
C08681=1087.347,312.222,413.367,176.705,23.642,153.740
C08682=1087.353,312.470,413.334,176.707,23.646,153.740
C08683=1087.358,312.718,413.304,176.710,23.650,153.741
C08684=1087.364,312.966,413.272,176.713,23.653,153.741
C08685=1087.370,313.214,413.240,176.716,23.657,153.742
C08686=1087.376,313.462,413.208,176.720,23.661,153.742
C08687=1087.382,313.710,413.176,176.723,23.664,153.742
C08688=1087.388,313.957,413.145,176.726,23.668,153.743
C08689=1087.394,314.206,413.113,176.729,23.672,153.743
C08690=1087.399,314.453,413.082,176.732,23.675,153.744
C08691=1087.405,314.701,413.050,176.735,23.679,153.744
C08692=1087.412,314.949,413.018,176.737,23.683,153.745
C08693=1087.417,315.197,412.987,176.740,23.687,153.745
C08694=1087.423,315.445,412.954,176.743,23.690,153.745
C08695=1087.428,315.693,412.922,176.747,23.695,153.746
C08696=1087.434,315.941,412.890,176.750,23.698,153.746
C08697=1087.443,316.345,412.838,176.754,23.704,153.747
C08698=1087.452,316.750,412.786,176.759,23.711,153.748
C08699=1087.461,317.154,412.734,176.764,23.717,153.749
C08700=1087.471,317.559,412.681,176.769,23.724,153.750
C08701=1087.476,317.806,412.649,176.772,23.727,153.750
C08702=1087.482,318.054,412.617,176.775,23.731,153.751
C08703=1087.488,318.303,412.585,176.778,23.735,153.751
C08704=1087.494,318.549,412.553,176.781,23.739,153.751
C08705=1087.499,318.798,412.520,176.784,23.743,153.752
C08706=1087.504,319.045,412.489,176.786,23.747,153.752
C08707=1087.510,319.294,412.457,176.790,23.751,153.753
C08708=1087.517,319.541,412.424,176.793,23.755,153.753
C08709=1087.522,319.789,412.392,176.796,23.758,153.754
C08710=1087.527,320.037,412.360,176.799,23.762,153.754
C08711=1087.533,320.286,412.328,176.802,23.766,153.755
C08712=1087.539,320.532,412.295,176.804,23.770,153.755
C08713=1087.545,320.781,412.263,176.808,23.774,153.756
C08714=1087.550,321.029,412.231,176.811,23.778,153.756
C08715=1087.556,321.276,412.198,176.814,23.782,153.757
C08716=1087.562,321.524,412.166,176.817,23.786,153.757
C08717=1087.568,321.772,412.133,176.820,23.789,153.758
C08718=1087.573,322.020,412.101,176.822,23.794,153.758
C08719=1087.579,322.267,412.068,176.826,23.798,153.759
C08720=1087.585,322.515,412.036,176.829,23.802,153.759
C08721=1087.591,322.764,412.004,176.832,23.806,153.760
C08722=1087.597,323.012,411.971,176.835,23.809,153.760
C08723=1087.602,323.259,411.939,176.837,23.813,153.761
C08724=1087.608,323.507,411.907,176.841,23.818,153.761
C08725=1087.614,323.755,411.873,176.844,23.821,153.762
C08726=1087.620,324.003,411.841,176.847,23.826,153.762
C08727=1087.626,324.250,411.809,176.850,23.829,153.763
C08728=1087.631,324.498,411.776,176.853,23.833,153.763
C08729=1087.637,324.746,411.743,176.856,23.838,153.764
C08730=1087.643,324.994,411.711,176.859,23.841,153.764
C08731=1087.649,325.242,411.678,176.862,23.845,153.765
C08732=1087.655,325.490,411.645,176.865,23.849,153.765
C08733=1087.660,325.737,411.614,176.868,23.853,153.766
C08734=1087.666,325.985,411.580,176.871,23.857,153.766
C08735=1087.672,326.233,411.548,176.874,23.862,153.767
C08736=1087.678,326.480,411.515,176.877,23.865,153.767
C08737=1087.684,326.729,411.482,176.880,23.869,153.768
C08738=1087.690,326.976,411.450,176.883,23.873,153.768
C08739=1087.696,327.224,411.417,176.887,23.877,153.769
C08740=1087.702,327.472,411.383,176.889,23.881,153.769
C08741=1087.708,327.720,411.351,176.892,23.885,153.770
C08742=1087.713,327.967,411.318,176.895,23.889,153.771
C08743=1087.719,328.215,411.286,176.899,23.893,153.771
C08744=1087.725,328.463,411.252,176.902,23.898,153.772
C08745=1087.731,328.710,411.220,176.904,23.902,153.772
C08746=1087.737,328.958,411.188,176.907,23.906,153.773
C08747=1087.742,329.206,411.154,176.911,23.910,153.773
C08748=1087.749,329.454,411.121,176.914,23.914,153.774
C08749=1087.758,329.851,411.068,176.919,23.920,153.775
C08750=1087.768,330.249,411.015,176.924,23.927,153.775
C08751=1087.777,330.647,410.963,176.928,23.933,153.776
C08752=1087.787,331.044,410.909,176.933,23.940,153.777
C08753=1087.793,331.292,410.876,176.937,23.944,153.778
C08754=1087.799,331.540,410.843,176.939,23.948,153.778
C08755=1087.805,331.788,410.810,176.942,23.952,153.779
C08756=1087.811,332.035,410.777,176.945,23.956,153.779
C08757=1087.817,332.283,410.743,176.949,23.961,153.780
C08758=1087.822,332.531,410.710,176.952,23.965,153.780
C08759=1087.829,332.779,410.677,176.954,23.969,153.781
C08760=1087.834,333.027,410.644,176.958,23.973,153.781
C08761=1087.840,333.275,410.611,176.961,23.978,153.782
C08762=1087.845,333.522,410.577,176.963,23.982,153.783
C08763=1087.852,333.769,410.544,176.966,23.986,153.783
C08764=1087.857,334.017,410.511,176.970,23.991,153.784
C08765=1087.863,334.265,410.477,176.973,23.995,153.784
C08766=1087.868,334.513,410.444,176.975,23.999,153.785
C08767=1087.874,334.760,410.410,176.979,24.004,153.786
C08768=1087.881,335.008,410.377,176.982,24.008,153.786
C08769=1087.886,335.256,410.344,176.985,24.012,153.787
C08770=1087.892,335.504,410.310,176.988,24.016,153.787
C08771=1087.898,335.751,410.276,176.991,24.021,153.788
C08772=1087.903,335.999,410.243,176.994,24.025,153.789
C08773=1087.909,336.247,410.210,176.998,24.029,153.789
C08774=1087.915,336.494,410.176,177.000,24.034,153.790
C08775=1087.921,336.742,410.143,177.003,24.038,153.790
C08776=1087.927,336.990,410.109,177.007,24.042,153.791
C08777=1087.933,337.238,410.075,177.010,24.046,153.791
C08778=1087.938,337.486,410.042,177.012,24.051,153.792
C08779=1087.945,337.733,410.008,177.016,24.055,153.793
C08780=1087.951,337.980,409.975,177.019,24.059,153.793
C08781=1087.956,338.228,409.941,177.021,24.064,153.794
C08782=1087.962,338.476,409.908,177.025,24.068,153.794
C08783=1087.968,338.724,409.873,177.028,24.073,153.795
C08784=1087.974,338.972,409.840,177.031,24.077,153.796
C08785=1087.980,339.219,409.806,177.034,24.082,153.796
C08786=1087.985,339.467,409.772,177.037,24.086,153.797
C08787=1087.991,339.714,409.738,177.040,24.091,153.798
C08788=1087.997,339.961,409.704,177.043,24.095,153.798
C08789=1088.003,340.209,409.671,177.046,24.099,153.799
C08790=1088.009,340.457,409.637,177.049,24.104,153.800
C08791=1088.015,340.704,409.603,177.052,24.108,153.800
C08792=1088.021,340.952,409.569,177.056,24.113,153.801
C08793=1088.026,341.200,409.535,177.059,24.117,153.801
C08794=1088.032,341.447,409.501,177.061,24.122,153.802
C08795=1088.038,341.696,409.467,177.065,24.127,153.803
C08796=1088.044,341.943,409.433,177.068,24.131,153.803
C08797=1088.049,342.190,409.399,177.071,24.136,153.804
C08798=1088.055,342.438,409.365,177.074,24.140,153.805
C08799=1088.061,342.686,409.331,177.077,24.144,153.805
C08800=1088.067,342.934,409.297,177.080,24.149,153.806
C08801=1088.077,343.325,409.243,177.085,24.156,153.807
C08802=1088.085,343.717,409.189,177.090,24.163,153.808
C08803=1088.095,344.109,409.135,177.095,24.170,153.809
C08804=1088.105,344.501,409.080,177.100,24.178,153.810
C08805=1088.110,344.748,409.046,177.103,24.182,153.811
C08806=1088.116,344.995,409.012,177.106,24.187,153.811
C08807=1088.123,345.243,408.978,177.109,24.192,153.812
C08808=1088.128,345.491,408.943,177.112,24.196,153.813
C08809=1088.134,345.738,408.909,177.115,24.201,153.813
C08810=1088.140,345.986,408.875,177.118,24.205,153.814
C08811=1088.146,346.233,408.841,177.121,24.210,153.815
C08812=1088.151,346.481,408.806,177.124,24.215,153.816
C08813=1088.158,346.729,408.772,177.127,24.220,153.816
C08814=1088.163,346.976,408.738,177.130,24.224,153.817
C08815=1088.169,347.224,408.703,177.134,24.229,153.818
C08816=1088.175,347.472,408.669,177.136,24.234,153.818
C08817=1088.181,347.719,408.635,177.140,24.239,153.819
C08818=1088.186,347.967,408.600,177.143,24.243,153.820
C08819=1088.192,348.215,408.565,177.146,24.248,153.820
C08820=1088.198,348.462,408.530,177.149,24.253,153.821
C08821=1088.204,348.709,408.496,177.152,24.258,153.822
C08822=1088.210,348.957,408.462,177.155,24.262,153.822
C08823=1088.215,349.204,408.427,177.159,24.267,153.823
C08824=1088.222,349.452,408.392,177.161,24.272,153.824
C08825=1088.227,349.699,408.357,177.165,24.277,153.825
C08826=1088.233,349.947,408.323,177.167,24.282,153.825
C08827=1088.240,350.195,408.289,177.171,24.286,153.826
C08828=1088.245,350.442,408.253,177.174,24.291,153.827
C08829=1088.251,350.690,408.219,177.177,24.296,153.828
C08830=1088.257,350.937,408.184,177.180,24.301,153.828
C08831=1088.263,351.185,408.149,177.183,24.306,153.829
C08832=1088.268,351.432,408.115,177.186,24.311,153.830
C08833=1088.275,351.679,408.080,177.189,24.316,153.830
C08834=1088.280,351.927,408.045,177.192,24.320,153.831
C08835=1088.287,352.174,408.010,177.196,24.325,153.832
C08836=1088.292,352.422,407.975,177.198,24.330,153.833
C08837=1088.298,352.669,407.940,177.202,24.335,153.833
C08838=1088.304,352.917,407.905,177.204,24.340,153.834
C08839=1088.310,353.164,407.870,177.208,24.345,153.835
C08840=1088.316,353.412,407.835,177.211,24.350,153.836
C08841=1088.322,353.659,407.801,177.214,24.354,153.836
C08842=1088.328,353.907,407.766,177.217,24.359,153.837
C08843=1088.333,354.154,407.730,177.220,24.365,153.838
C08844=1088.340,354.402,407.696,177.224,24.370,153.839
C08845=1088.345,354.649,407.660,177.226,24.375,153.839
C08846=1088.351,354.897,407.625,177.230,24.380,153.840
C08847=1088.357,355.144,407.591,177.232,24.384,153.841
C08848=1088.363,355.392,407.555,177.236,24.390,153.842
C08849=1088.369,355.639,407.520,177.238,24.395,153.843
C08850=1088.374,355.887,407.485,177.242,24.400,153.843
C08851=1088.381,356.134,407.449,177.245,24.405,153.844
C08852=1088.387,356.381,407.414,177.248,24.410,153.845
C08853=1088.396,356.776,407.358,177.253,24.418,153.846
C08854=1088.405,357.170,407.302,177.258,24.426,153.847
C08855=1088.415,357.564,407.245,177.263,24.434,153.849
C08856=1088.424,357.959,407.190,177.268,24.443,153.850
C08857=1088.430,358.207,407.154,177.271,24.447,153.851
C08858=1088.436,358.455,407.118,177.275,24.453,153.852
C08859=1088.442,358.701,407.083,177.277,24.458,153.852
C08860=1088.448,358.949,407.048,177.281,24.463,153.853
C08861=1088.454,359.197,407.012,177.283,24.468,153.854
C08862=1088.460,359.444,406.977,177.287,24.473,153.855
C08863=1088.466,359.691,406.941,177.290,24.479,153.856
C08864=1088.473,359.939,406.906,177.293,24.484,153.856
C08865=1088.478,360.186,406.870,177.296,24.489,153.857
C08866=1088.484,360.433,406.835,177.299,24.494,153.858
C08867=1088.490,360.681,406.799,177.302,24.500,153.859
C08868=1088.496,360.928,406.763,177.305,24.505,153.860
C08869=1088.502,361.176,406.728,177.308,24.510,153.861
C08870=1088.508,361.423,406.692,177.312,24.515,153.862
C08871=1088.513,361.670,406.656,177.315,24.521,153.862
C08872=1088.519,361.917,406.620,177.317,24.526,153.863
C08873=1088.525,362.165,406.584,177.321,24.531,153.864
C08874=1088.531,362.412,406.549,177.324,24.537,153.865
C08875=1088.537,362.660,406.513,177.327,24.542,153.866
C08876=1088.543,362.907,406.477,177.330,24.547,153.867
C08877=1088.549,363.154,406.441,177.334,24.553,153.867
C08878=1088.555,363.401,406.406,177.336,24.558,153.868
C08879=1088.561,363.649,406.370,177.340,24.563,153.869
C08880=1088.567,363.896,406.334,177.343,24.569,153.870
C08881=1088.573,364.144,406.298,177.346,24.574,153.871
C08882=1088.578,364.391,406.263,177.349,24.580,153.872
C08883=1088.585,364.638,406.226,177.352,24.585,153.873
C08884=1088.591,364.885,406.190,177.355,24.591,153.874
C08885=1088.597,365.133,406.155,177.358,24.596,153.875
C08886=1088.603,365.380,406.118,177.362,24.602,153.875
C08887=1088.609,365.627,406.083,177.364,24.607,153.876
C08888=1088.615,365.874,406.046,177.367,24.613,153.877
C08889=1088.620,366.122,406.010,177.371,24.618,153.878
C08890=1088.627,366.369,405.974,177.374,24.624,153.879
C08891=1088.632,366.616,405.938,177.377,24.629,153.880
C08892=1088.638,366.863,405.902,177.380,24.635,153.881
C08893=1088.644,367.111,405.866,177.383,24.641,153.882
C08894=1088.650,367.358,405.829,177.386,24.646,153.883
C08895=1088.656,367.605,405.793,177.389,24.652,153.884
C08896=1088.662,367.852,405.757,177.393,24.658,153.885
C08897=1088.668,368.099,405.721,177.396,24.663,153.886
C08898=1088.673,368.347,405.684,177.398,24.669,153.887
C08899=1088.680,368.594,405.648,177.402,24.674,153.888
C08900=1088.686,368.841,405.612,177.405,24.680,153.889
C08901=1088.691,369.089,405.575,177.408,24.686,153.889
C08902=1088.698,369.336,405.539,177.411,24.691,153.890
C08903=1088.703,369.583,405.503,177.414,24.697,153.891
C08904=1088.709,369.830,405.466,177.418,24.703,153.892
C08905=1088.719,370.240,405.405,177.423,24.712,153.894
C08906=1088.729,370.650,405.345,177.428,24.722,153.896
C08907=1088.739,371.060,405.284,177.433,24.731,153.897
C08908=1088.750,371.471,405.224,177.438,24.741,153.899
C08909=1088.755,371.717,405.188,177.441,24.747,153.900
C08910=1088.761,371.965,405.151,177.444,24.753,153.901
C08911=1088.767,372.212,405.114,177.448,24.759,153.902
C08912=1088.773,372.459,405.077,177.451,24.764,153.903
C08913=1088.779,372.706,405.041,177.453,24.770,153.904
C08914=1088.786,372.953,405.004,177.457,24.776,153.905
C08915=1088.791,373.201,404.967,177.460,24.782,153.906
C08916=1088.798,373.448,404.931,177.463,24.788,153.907
C08917=1088.804,373.695,404.894,177.467,24.794,153.908
C08918=1088.810,373.942,404.857,177.469,24.800,153.909
C08919=1088.816,374.190,404.820,177.472,24.805,153.910
C08920=1088.822,374.437,404.783,177.476,24.812,153.911
C08921=1088.827,374.684,404.747,177.479,24.818,153.912
C08922=1088.833,374.931,404.710,177.482,24.824,153.913
C08923=1088.839,375.178,404.673,177.486,24.830,153.914
C08924=1088.846,375.425,404.636,177.488,24.836,153.915
C08925=1088.851,375.672,404.599,177.491,24.842,153.916
C08926=1088.857,375.919,404.562,177.494,24.848,153.917
C08927=1088.864,376.167,404.525,177.498,24.854,153.918
C08928=1088.870,376.414,404.487,177.501,24.860,153.919
C08929=1088.875,376.661,404.450,177.504,24.866,153.920
C08930=1088.882,376.908,404.414,177.507,24.872,153.921
C08931=1088.887,377.155,404.376,177.510,24.878,153.922
C08932=1088.893,377.402,404.339,177.513,24.884,153.923
C08933=1088.899,377.650,404.303,177.516,24.891,153.924
C08934=1088.905,377.896,404.265,177.520,24.897,153.926
C08935=1088.911,378.144,404.228,177.523,24.903,153.927
C08936=1088.917,378.391,404.191,177.526,24.909,153.928
C08937=1088.923,378.637,404.154,177.529,24.916,153.929
C08938=1088.929,378.885,404.117,177.532,24.922,153.930
C08939=1088.936,379.132,404.079,177.535,24.928,153.931
C08940=1088.942,379.379,404.042,177.538,24.934,153.932
C08941=1088.948,379.626,404.004,177.541,24.940,153.933
C08942=1088.953,379.873,403.967,177.545,24.947,153.934
C08943=1088.960,380.120,403.930,177.548,24.953,153.936
C08944=1088.966,380.367,403.892,177.551,24.959,153.937
C08945=1088.972,380.615,403.855,177.554,24.966,153.938
C08946=1088.978,380.861,403.817,177.557,24.972,153.939
C08947=1088.984,381.108,403.780,177.561,24.979,153.940
C08948=1088.990,381.355,403.743,177.564,24.985,153.941
C08949=1088.996,381.602,403.705,177.567,24.991,153.942
C08950=1089.002,381.849,403.667,177.569,24.997,153.943
C08951=1089.009,382.096,403.631,177.572,25.004,153.945
C08952=1089.015,382.343,403.593,177.576,25.011,153.946
C08953=1089.021,382.590,403.555,177.579,25.017,153.947
C08954=1089.027,382.837,403.517,177.582,25.023,153.948
C08955=1089.033,383.085,403.480,177.585,25.030,153.949
C08956=1089.039,383.331,403.442,177.588,25.037,153.950
C08957=1089.044,383.550,403.409,177.592,25.042,153.951
C08958=1089.049,383.769,403.375,177.594,25.048,153.952
C08959=1089.055,383.988,403.342,177.596,25.054,153.954
C08960=1089.060,384.207,403.309,177.600,25.060,153.955
C08961=1089.065,384.426,403.275,177.602,25.066,153.956
C08962=1089.071,384.645,403.241,177.606,25.072,153.957
C08963=1089.076,384.864,403.207,177.608,25.078,153.958
C08964=1089.081,385.083,403.174,177.611,25.084,153.959
C08965=1089.087,385.330,403.136,177.614,25.090,153.960
C08966=1089.093,385.577,403.098,177.618,25.097,153.961
C08967=1089.099,385.823,403.061,177.621,25.104,153.962
C08968=1089.106,386.071,403.023,177.624,25.111,153.964
C08969=1089.112,386.318,402.985,177.627,25.117,153.965
C08970=1089.118,386.564,402.947,177.630,25.124,153.966
C08971=1089.124,386.812,402.909,177.633,25.131,153.967
C08972=1089.129,387.059,402.871,177.636,25.138,153.969
C08973=1089.135,387.305,402.832,177.639,25.144,153.970
C08974=1089.142,387.552,402.794,177.643,25.151,153.971
C08975=1089.148,387.799,402.756,177.646,25.158,153.973
C08976=1089.154,388.046,402.718,177.649,25.165,153.974
C08977=1089.160,388.293,402.680,177.652,25.172,153.975
C08978=1089.166,388.540,402.642,177.655,25.179,153.976
C08979=1089.172,388.786,402.604,177.658,25.186,153.978
C08980=1089.178,389.034,402.565,177.661,25.192,153.979
C08981=1089.184,389.280,402.527,177.664,25.199,153.980
C08982=1089.191,389.528,402.489,177.667,25.206,153.981
C08983=1089.197,389.774,402.451,177.670,25.213,153.983
C08984=1089.204,390.021,402.412,177.674,25.221,153.984
C08985=1089.210,390.268,402.374,177.678,25.227,153.985
C08986=1089.216,390.515,402.335,177.681,25.234,153.987
C08987=1089.221,390.762,402.297,177.684,25.241,153.988
C08988=1089.228,391.009,402.259,177.687,25.248,153.989
C08989=1089.234,391.255,402.221,177.690,25.255,153.990
C08990=1089.241,391.503,402.183,177.693,25.262,153.992
C08991=1089.246,391.749,402.143,177.696,25.269,153.993
C08992=1089.253,391.997,402.105,177.699,25.276,153.994
C08993=1089.259,392.243,402.067,177.703,25.284,153.996
C08994=1089.265,392.490,402.027,177.706,25.291,153.997
C08995=1089.271,392.737,401.990,177.709,25.298,153.999
C08996=1089.278,392.984,401.951,177.712,25.305,154.000
C08997=1089.283,393.231,401.912,177.715,25.313,154.001
C08998=1089.290,393.477,401.874,177.718,25.320,154.003
C08999=1089.296,393.725,401.834,177.721,25.327,154.004
C09000=1089.302,393.971,401.796,177.725,25.335,154.005
C09001=1089.308,394.218,401.757,177.728,25.342,154.007
C09002=1089.314,394.465,401.719,177.731,25.349,154.008
C09003=1089.320,394.712,401.679,177.734,25.357,154.010
C09004=1089.327,394.959,401.641,177.737,25.364,154.011
C09005=1089.333,395.205,401.603,177.740,25.371,154.012
C09006=1089.339,395.452,401.563,177.744,25.379,154.014
C09007=1089.344,395.699,401.524,177.747,25.386,154.015
C09008=1089.351,395.946,401.485,177.750,25.394,154.017
C09009=1089.357,396.193,401.446,177.753,25.401,154.018
C09010=1089.363,396.440,401.408,177.756,25.408,154.019
C09011=1089.369,396.687,401.369,177.760,25.416,154.021
C09012=1089.375,396.934,401.329,177.763,25.424,154.022
C09013=1089.381,397.159,401.293,177.765,25.431,154.024
C09014=1089.387,397.384,401.258,177.768,25.438,154.025
C09015=1089.392,397.611,401.222,177.771,25.445,154.026
C09016=1089.398,397.836,401.186,177.774,25.452,154.028
C09017=1089.404,398.061,401.151,177.777,25.459,154.029
C09018=1089.409,398.287,401.114,177.780,25.465,154.030
C09019=1089.415,398.513,401.079,177.783,25.473,154.032
C09020=1089.421,398.739,401.043,177.786,25.480,154.033
C09021=1089.427,398.985,401.004,177.789,25.488,154.035
C09022=1089.433,399.232,400.965,177.792,25.495,154.036
C09023=1089.440,399.479,400.925,177.796,25.503,154.038
C09024=1089.446,399.726,400.886,177.798,25.511,154.039
C09025=1089.452,399.973,400.846,177.801,25.518,154.041
C09026=1089.457,400.219,400.807,177.805,25.527,154.042
C09027=1089.463,400.466,400.768,177.808,25.535,154.044
C09028=1089.470,400.713,400.728,177.811,25.542,154.045
C09029=1089.477,400.960,400.689,177.814,25.550,154.047
C09030=1089.483,401.207,400.649,177.818,25.559,154.048
C09031=1089.489,401.453,400.610,177.821,25.566,154.050
C09032=1089.495,401.700,400.570,177.824,25.574,154.052
C09033=1089.501,401.947,400.531,177.827,25.582,154.053
C09034=1089.507,402.193,400.491,177.830,25.590,154.055
C09035=1089.513,402.441,400.451,177.833,25.598,154.056
C09036=1089.520,402.687,400.412,177.837,25.607,154.058
C09037=1089.526,402.934,400.372,177.840,25.615,154.059
C09038=1089.532,403.181,400.333,177.843,25.623,154.061
C09039=1089.539,403.428,400.293,177.847,25.631,154.063
C09040=1089.544,403.674,400.254,177.849,25.639,154.064
C09041=1089.551,403.921,400.213,177.853,25.647,154.066
C09042=1089.557,404.168,400.174,177.856,25.656,154.068
C09043=1089.563,404.414,400.134,177.859,25.663,154.069
C09044=1089.569,404.661,400.094,177.863,25.672,154.071
C09045=1089.576,404.908,400.054,177.865,25.680,154.072
C09046=1089.582,405.154,400.014,177.869,25.689,154.074
C09047=1089.588,405.401,399.974,177.872,25.697,154.076
C09048=1089.594,405.648,399.935,177.875,25.705,154.077
C09049=1089.601,405.894,399.894,177.879,25.714,154.079
C09050=1089.607,406.141,399.854,177.881,25.722,154.081
C09051=1089.613,406.388,399.815,177.885,25.730,154.082
C09052=1089.620,406.635,399.775,177.888,25.739,154.084
C09053=1089.625,406.881,399.734,177.892,25.748,154.086
C09054=1089.632,407.128,399.694,177.895,25.756,154.088
C09055=1089.638,407.375,399.654,177.898,25.765,154.089
C09056=1089.644,407.621,399.614,177.901,25.773,154.091
C09057=1089.651,407.868,399.573,177.905,25.782,154.093
C09058=1089.657,408.115,399.534,177.908,25.790,154.094
C09059=1089.662,408.362,399.493,177.911,25.799,154.096
C09060=1089.669,408.608,399.453,177.914,25.808,154.098
C09061=1089.676,408.855,399.413,177.918,25.817,154.100
C09062=1089.681,409.102,399.372,177.920,25.825,154.101
C09063=1089.688,409.349,399.332,177.924,25.834,154.103
C09064=1089.694,409.595,399.292,177.927,25.843,154.105
C09065=1089.700,409.841,399.250,177.931,25.852,154.107
C09066=1089.707,410.088,399.210,177.934,25.861,154.109
C09067=1089.713,410.334,399.170,177.937,25.869,154.110
C09068=1089.719,410.581,399.129,177.941,25.879,154.112
C09069=1089.724,410.807,399.092,177.944,25.887,154.114
C09070=1089.730,411.033,399.055,177.946,25.895,154.115
C09071=1089.737,411.260,399.018,177.949,25.903,154.117
C09072=1089.742,411.486,398.980,177.952,25.912,154.119
C09073=1089.748,411.713,398.943,177.955,25.919,154.120
C09074=1089.754,411.938,398.906,177.959,25.928,154.122
C09075=1089.759,412.165,398.869,177.962,25.937,154.124
C09076=1089.765,412.391,398.831,177.965,25.945,154.126
C09077=1089.772,412.637,398.791,177.967,25.954,154.127
C09078=1089.778,412.884,398.749,177.971,25.963,154.129
C09079=1089.784,413.131,398.709,177.975,25.972,154.131
C09080=1089.790,413.377,398.668,177.977,25.981,154.133
C09081=1089.797,413.624,398.627,177.981,25.991,154.135
C09082=1089.803,413.871,398.586,177.985,26.000,154.137
C09083=1089.810,414.117,398.546,177.988,26.009,154.139
C09084=1089.816,414.363,398.505,177.991,26.018,154.141
C09085=1089.823,414.610,398.464,177.994,26.028,154.143
C09086=1089.829,414.857,398.423,177.998,26.037,154.144
C09087=1089.835,415.103,398.382,178.001,26.046,154.146
C09088=1089.842,415.349,398.341,178.004,26.056,154.148
C09089=1089.848,415.596,398.300,178.008,26.065,154.150
C09090=1089.855,415.843,398.259,178.012,26.075,154.152
C09091=1089.861,416.089,398.217,178.014,26.084,154.154
C09092=1089.868,416.336,398.177,178.018,26.094,154.156
C09093=1089.874,416.582,398.135,178.021,26.103,154.158
C09094=1089.880,416.829,398.094,178.025,26.113,154.160
C09095=1089.886,417.075,398.052,178.028,26.123,154.162
C09096=1089.893,417.322,398.012,178.031,26.132,154.164
C09097=1089.899,417.568,397.970,178.035,26.142,154.166
C09098=1089.905,417.814,397.929,178.038,26.152,154.168
C09099=1089.912,418.061,397.888,178.042,26.162,154.170
C09100=1089.918,418.307,397.846,178.045,26.171,154.172
C09101=1089.925,418.554,397.804,178.048,26.181,154.174
C09102=1089.931,418.800,397.763,178.051,26.191,154.176
C09103=1089.938,419.047,397.722,178.055,26.201,154.179
C09104=1089.944,419.293,397.680,178.058,26.211,154.180
C09105=1089.950,419.539,397.639,178.062,26.221,154.183
C09106=1089.956,419.786,397.597,178.065,26.231,154.185
